// TwinCAT 3 PLC project DPPLC
// Title: YK_DPJ
// Company: YK
// Author: DHW
// ProjectVersion: V1.1
// ProgramVersion: 3.1.4023.0
// CompilerDefines: VISU_USEWSTRING
// libraries:
//   Lib_Basic, * (Beckhoff_GZ)
//   Lib_FileOperation, * (Beckhoff_GZ)
//   Tc2_EtherCAT, * (Beckhoff Automation GmbH)
//   Tc2_Math, * (Beckhoff Automation GmbH)
//   Tc2_MC2, * (Beckhoff Automation GmbH)
//   Tc2_MC2_Camming, * (Beckhoff Automation GmbH)
//   Tc2_MC2_FlyingSaw, * (Beckhoff Automation GmbH)
//   Tc2_Standard, * (Beckhoff Automation GmbH)
//   Tc2_System, * (Beckhoff Automation GmbH)
//   Tc2_TcpIp, * (Beckhoff Automation GmbH)
//   Tc2_Utilities, * (Beckhoff Automation GmbH)
//   Tc2_XmlDataSrv, * (Beckhoff Automation GmbH)
//   Tc3_MC2_AdvancedHoming, * (Beckhoff Automation GmbH)
//   Tc3_Module, * (Beckhoff Automation GmbH)
//   VisuDialogs, * (System)
//   VisuElemEventTable, * (System)
//   VisuSymbols, * (System)
//   VisuSymbols,3.5.10.0,System
// project tree:
//   P2DUTs/01_AxisCO_Ntrol/ MC_AxisParameter.TcDUT, ST_Dust_Motor.TcDUT, ST_ECYCtrl.TcDUT, ST_JXCE.TcDUT, ST_SetpMotor.TcDUT
//   P2DUTs/01_AxisCO_Ntrol_1/ ST_AxisCmd.TcDUT, ST_AxisCtrl.TcDUT, ST_AxisIo.TcDUT, ST_AxisStatus.TcDUT, ST_Axis_Par.TcDUT
//   P2DUTs/02_Cylinder/ ST_CyCmd.TcDUT, ST_CyCtrl.TcDUT, ST_CYIo.TcDUT, ST_CyStatus.TcDUT
//   P2DUTs/06_Interface/FB_Interface/ ST_Cam.TcDUT, ST_Gear.TcDUT, ST_GearInPos.TcDUT, ST_Tension.TcDUT
//   P2DUTs/06_Interface/ IData.TcDUT, IM2Glue.TcDUT
//   P2DUTs/06_Interface/Method/ ST_Method.TcDUT, ST_MethodOut.TcDUT
//   P2DUTs/07_Name/ ST_Dust.TcDUT, ST_AxisName.TcDUT, ST_CylinderName.TcDUT, ST_ElectValveName.TcDUT, ST_P2AxisName.TcDUT, ST_P2CylinderName.TcDUT, ST_P2ElectValveName.TcDUT, ST_P2VirAxisName.TcDUT, ST_RecName.TcDUT, ST_TableName.TcDUT, ST_VirAxisName.TcDUT
//   P2DUTs/08_IO/ ST_Button.TcDUT, ST_P2Button.TcDUT, ST_P2Senser.TcDUT, ST_Senser.TcDUT, ST_SystemButton.TcDUT, System_Senser.TcDUT
//   P2DUTs/30_Parameter/04_Rectify/ ST_PLC_PC_MES.TcDUT, ST_RecCmd.TcDUT, ST_RecCtrl.TcDUT, ST_RecIo.TcDUT, ST_RecStatus.TcDUT
//   P2DUTs/30_Parameter/ ST_DT_To_MQ_MES.TcDUT, ST_MQ_To_DT_MES.TcDUT, ST_ParFilterAD.TcDUT, ST_ParMachine.TcDUT, ST_ParProduct.TcDUT, ST_ParTableNo.TcDUT
//   P2DUTs/31_其他辅助/ DToM_Process.TcDUT, DToM_System.TcDUT, File_com_typ.TcDUT, MToD_Process.TcDUT, MToD_System.TcDUT, ST_DATA_NEED_BE_PERSIS.TcDUT
//   P2DUTs/32_系统/ IModeEN.TcDUT, IRecipe.TcDUT, ST_SysCmd.TcDUT, ST_SystemRUN.TcDUT
//   P2DUTs/33_M2/ ST_BeltData.TcDUT, ST_BeltData1.TcDUT
//   P2DUTs/34_M1/ ST_Rectify.TcDUT
//   P2DUTs/35_CCD/35_CCD/ ICCD_1.TcDUT, STCcdData_1.TcDUT, ST_CCDCom.TcDUT, ST_CCDComOverhang.TcDUT, ST_CCDComRectify.TcDUT, ST_CCDComRectify_I.TcDUT, ST_CCDComRectify_O.TcDUT, ST_CCDOverhang_I.TcDUT, ST_CCDOverhang_O.TcDUT, ST_Ng_classification.TcDUT
//   P2DUTs/35_CCD/ ICCD.TcDUT, STCcdData.TcDUT, STCcdDataSend.TcDUT
//   P2DUTs/36_ShortTest/ CMD.TcDUT, IShortTest.TcDUT, ShortDataShow.TcDUT, ShortPar.TcDUT
//   P2DUTs/37_Code/ ICode.TcDUT, ParCode.TcDUT
//   P2DUTs/38_User1/ ControlSignal.TcDUT, EleControlNo.TcDUT, LocalProduction.TcDUT, P2_AxiseNo.TcDUT, P2_TableNo.TcDUT, Parameters.TcDUT, sMC_CAM_REF.TcDUT, System_Control.TcDUT, User1_Par.TcDUT
//   P2DUTs/39User2/ conAn_date.TcDUT, conCa_date.TcDUT, conDT_Date.TcDUT, conDT_RunStatus.TcDUT, conStickGlue_date.TcDUT, conTailCurl_date.TcDUT, parDT_date.TcDUT, parMechanical.TcDUT, parTailCurl_date.TcDUT, Scan_TJ.TcDUT, ST_Timedata.TcDUT, ST_Torque.TcDUT, ST_UserControl.TcDUT
//   P2DUTs/指纹/ ST_FingerprintKey.TcDUT
//   P2GVLs/ GCylinder.TcGVL, GMotion.TcGVL, GVL_Par.TcGVL, GVL_User2.TcGVL, GVL_User3.TcGVL, IO.TcGVL, N.TcGVL, System.TcGVL, User01.TcGVL
//   P2POUs/BasicFunction/01_IO/ FB_Filter_AD.TcPOU (encrypted, skipped), FB_Filter_ADV2.TcPOU (encrypted, skipped), FB_RotateSwitchCode.TcPOU (encrypted, skipped), ScaleTrans.TcPOU, ScaleTrans_1.TcPOU
//   P2POUs/BasicFunction/02_SystemCheck/ CheckBounds.TcPOU, CheckDivDInt.TcPOU, CheckDivLInt.TcPOU, CheckDivLReal.TcPOU, CheckDivReal.TcPOU, CheckLRangeSigned.TcPOU, CheckLRangeUnsigned.TcPOU, CheckPointer.TcPOU, CheckRangeSigned.TcPOU, CheckRangeUnsigned.TcPOU
//   P2POUs/BasicFunction/03_Motion/ Ax_FindHomeV3.TcPOU (encrypted, skipped), CS_AxisCtrl.TcPOU, CS_DustMoter.TcPOU, CS_SetpMoter.TcPOU, Three_Scale.TcPOU
//   P2POUs/BasicFunction/04_Gear/ FB_GearInDyn.TcPOU (encrypted, skipped), FB_GearInMulti.TcPOU (encrypted, skipped), FB_GearInPos.TcPOU (encrypted, skipped)
//   P2POUs/BasicFunction/05_Actuators/ FB_Cylinder.TcPOU, FB_CylinderV2.TcPOU, FB_Vacuum.TcPOU
//   P2POUs/BasicFunction/06_Public/ FC_AngleToLength.TcPOU (encrypted, skipped), FC_LengthToAngle.TcPOU (encrypted, skipped), f_Length2.TcPOU (encrypted, skipped), f_Length2_1.TcPOU (encrypted, skipped), PulseCtrl.TcPOU (encrypted, skipped), PulseGeneratorCtrl.TcPOU (encrypted, skipped)
//   P2POUs/BasicFunction/07_Ten/ FB_TensionGM.TcPOU (encrypted, skipped), FB_TensionGMV2.TcPOU (encrypted, skipped), FB_TensionGMV2_1.TcPOU (encrypted, skipped), FB_TensionGMV3.TcPOU (encrypted, skipped), FB_TensionP4Buffer.TcPOU (encrypted, skipped), FB_TensionPole.TcPOU (encrypted, skipped), FB_TensionV3.TcPOU (encrypted, skipped)
//   P2POUs/BasicFunction/08_Data/ CS_Data.TcPOU, CS_Data_Test.TcPOU, CS_Recipe.TcPOU, FB_DataXML.TcPOU, FB_DataXML_old.TcPOU, FB_DTData.TcPOU
//   P2POUs/BasicFunction/09_User1/ Dp_Roll_New.TcPOU (encrypted, skipped), Dp_Roll_New_BAK.TcPOU, Dp_Roll_V2.TcPOU, FB_CamIn.TcPOU (encrypted, skipped), FB_CamGMVir.TcPOU (encrypted, skipped), FB_CamPTPTest.TcPOU (encrypted, skipped), FB_CamPTPTestV2.TcPOU (encrypted, skipped), FB_CamTrapezoid.TcPOU (encrypted, skipped), FB_CreatCamEndWind.TcPOU (encrypted, skipped), FB_CreatCamGMBuffer.TcPOU (encrypted, skipped), FB_CreatCamVirGMDriver.TcPOU (encrypted, skipped), FB_CrectCamGMDanserMove.TcPOU (encrypted, skipped), FB_CrectCamMove.TcPOU, FB_CrectCamUpDown.TcPOU, FB_CrectCamUpDown_1.TcPOU, FB_CrectCamUpDown_10.TcPOU, FB_CrectCamUpDown_2.TcPOU, FB_CrectCamUpDown_3.TcPOU, FB_CrectCamUpDown_4.TcPOU, FB_CrectCamYaDaoLine.TcPOU, FB_CrectCamYaDaoLine2_V2.TcPOU, FB_CrectCamYaDaoLine_V2.TcPOU, FB_CrectCamYaDaoUpDown.TcPOU, FB_CrectCamYaDaoUpDown2.TcPOU, FB_GMLengthDown_L.TcPOU (encrypted, skipped), FB_GMLengthDown_R.TcPOU (encrypted, skipped), FB_GMLengthUp.TcPOU (encrypted, skipped), FB_GMLengthUp_L.TcPOU (encrypted, skipped), FB_GMLengthUp_R.TcPOU (encrypted, skipped), FB_RectifyGM.TcPOU (encrypted, skipped)
//   P2POUs/BasicFunction/10_MES/ CS_CcdTcp.TcPOU, CS_CcdTcp_V2.TcPOU, CS_CodeTcp.TcPOU, CS_FsyTcp.TcPOU
//   P2POUs/BasicFunction/11_SystemInfo/ SystemInfoCtrl.TcPOU, TaskInfoCtrl.TcPOU
//   P2POUs/BasicFunction/12_User2/ FB_AxisHandautomatic.TcPOU, FB_BlueFlag.TcPOU, FB_BlueGlue.TcPOU, FB_CamDTDriver.TcPOU, FB_Demarcate.TcPOU, FB_DiameterORLength.TcPOU, FB_RecdevPla.TcPOU, FB_Rectify.TcPOU, FB_RectifyTry.TcPOU, FB_SuckerTest.TcPOU, Program_1.TcPOU, Rectifydev_PID.TcPOU
//   P2POUs/POUS/ FingerprintKey.TcPOU, FunctionTest.TcPOU, IOLink.TcPOU, MAIN.TcPOU, MainState.TcPOU, P2M1_Auto.TcPOU, P2M2_Auto.TcPOU, P2M3_Auto.TcPOU, P2Program_FB.TcPOU
//   P3GVLs/ P3IO.TcGVL, P3Motion.TcGVL, P3Name.TcGVL, P3Par.TcGVL, P3Press.TcGVL, P3Temperature.TcGVL
//   P3POUs/P3FB/ ADSWrite_Limit.TcPOU, CS_AxisCtrlV2.TcPOU (encrypted, skipped), CS_SetpMoterV2.TcPOU, FB_AxisHandautomatic_1.TcPOU, FB_Blink.TcPOU, FB_CSP_Velo_Torque.TcPOU, FB_DataXMLP3.TcPOU, FB_DataXMLP3_Old.TcPOU, FB_HDData.TcPOU, FB_OEE.TcPOU, FB_Press.TcPOU, FB_ProductionDataLocal.TcPOU, FB_PulsPercentage.TcPOU, FB_Temperature.TcPOU, Oven_button.TcPOU, Oven_Time.TcPOU, FB_SetMoter_auto.TcPOU, Sampling.TcPOU, ShortTest.TcPOU, Unwinding_PID.TcPOU, Weight_cese.TcPOU
//   P3POUs/POUs/Auto%28PRG%29/ LateBlanking_Auto1.TcPOU (not stored), LateBlanking_Auto2.TcPOU (not stored), LateBlanking_Auto3.TcPOU (not stored), LateBlanking_Auto4.TcPOU (not stored), LateBlanking_Auto5.TcPOU (not stored), LateBlanking_Auto6.TcPOU (not stored), LateBlanking_Auto7.TcPOU (not stored), LateBlanking_Auto8_01Sticke.TcPOU (not stored), LateBlanking_Auto9_02Sticke.TcPOU (not stored), LateBlanking_Auto1_Stick.TcPOU (not stored)
//   P3POUs/POUs/Auxiliary/ LateBlankingCylinderManual.TcPOU, LateBlankingMotorManual.TcPOU, LateBlanking_Alarm.TcPOU, LateBlanking_Condition.TcPOU, LateBlanking_Scan.TcPOU, LateBlanking_Short_Test.TcPOU, LateBlanking_Temperature.TcPOU, LateBlanking_Thickness_Test.TcPOU, LateBlanking_Tips.TcPOU, LateBlanking_Weight_Test.TcPOU, MES_JT_ZT.TcPOU, MQ_FSY.TcPOU, Output_statistics.TcPOU
//   P3POUs/POUs/Init/ L_Init1.TcPOU, L_Init2.TcPOU, L_Init3.TcPOU, L_Init4.TcPOU, L_Init5.TcPOU, L_Init6.TcPOU, L_Init7.TcPOU, L_Init8.TcPOU
//   P3POUs/POUs/ P3IOLink.TcPOU, P3MAIN.TcPOU, P3MainState.TcPOU
//   P3UDTs/MES/ DTM_Mes1.TcDUT, Mes1.TcDUT, Mes2.TcDUT, MTD_Mes1.TcDUT
//   P3UDTs/Output_statistic/ Statistics.TcDUT, ST_Timedata_1.TcDUT
//   P3UDTs/P3_AxisCO_Ntrol/ ST_AxisCmdV2.TcDUT, ST_AxisCtrlV2.TcDUT, ST_Axis_ParV2.TcDUT
//   P3UDTs/P3_IO/ ST_P3Button.TcDUT, ST_P3Senser.TcDUT
//   P3UDTs/P3_Memory/ ST_CellMemory.TcDUT
//   P3UDTs/P3_Name/ ST_MemoryName.TcDUT, ST_P3AxisName.TcDUT, ST_P3CylinderName.TcDUT, ST_P3ElectValveName.TcDUT, ST_TempName.TcDUT
//   P3UDTs/P3_par/ P3_Par.TcDUT, User2_Par.TcDUT
//   P3UDTs/P3_ShortTest/ CMD_1.TcDUT, ShortCiucitCtrl.TcDUT, ShortDataShow_1.TcDUT, ShortPar_1.TcDUT, ShortTestCtrl.TcDUT, ShortTestReceiveData.TcDUT, ShortTestSendData.TcDUT, ST_ReceiveTestStatus.TcDUT, ST_SendTestStatus.TcDUT
//   P3UDTs/P3_Temperature/ STTempCtrl.TcDUT, ST_ParTemperature.TcDUT, TempIn.TcDUT, TempInShow.TcDUT, TempOut.TcDUT
//   P3UDTs/P3_Thickness/ ST_Thickness.TcDUT
//   P3UDTs/P3_Torque/ ST_TorqueMotion.TcDUT, ST_Torque_P3.TcDUT
//   P3UDTs/P3_Variable/ ST_StickIDGlue_date.TcDUT
//   P3UDTs/P3_Weight/ ST_Gross.TcDUT, ST_ReceiveData.TcDUT, ST_ReceiveStatus.TcDUT, ST_SendData.TcDUT, ST_SendStatus.TcDUT
//   / Task_P2M1.TcTTO, Task_P2M2.TcTTO, Task_P2M3.TcTTO, Task_P2Main.TcTTO, Task_P3.TcTTO
// real-time tasks:
//   TASK Task P1: cycle T#2ms, priority 8, ADS port 350
//   TASK Task P2M1: cycle T#2ms, priority 16, ADS port 351
//   TASK Task P3: cycle T#2ms, priority 18, ADS port 352
//   TASK Task P2M2: cycle T#2ms, priority 14, ADS port 353
//   TASK Task P2M3: cycle T#2ms, priority 12, ADS port 354
//   TASK Task P2Main: cycle T#2ms, priority 10, ADS port 355
// motion (NC):
//   TASK NC-Task 1 SAF: cycle T#2ms, priority 2, ADS port 501
//   TASK NC-Task 1 SVB: cycle T#2ms, priority 4, ADS port 511
//   AXIS Axis001_1 P1An_UnWind_L (id 1) // 正极模切左放卷
//     General: UnitName=°
//     Dynamic: Acceleration=6210, Deceleration=6210, Jerk=225521
//     Velo: SlowManual=20, FastManual=20, Maximum=450
//     OtherSettings: AllowMotionCmdToSlave=true
//     encoder EncType=19
//       EncPara: ScaleFactorNumerator=2.86102e-06, MaxCount=#xffffffff
//     drive DrvType=16
//       DrvPara: MaxCount=#xffffffff, DriveControlDWord=#x00020100
//         Analog: VeloReferenz=450, TorqueSetpointScale=10, ScaleFactorActTorque=0.1
//         TimeComp: TaskDelayCycles=1
//     controller CtrType=1
//       CtrPara: PriorControlFactor=1
//         PosDiffControl: Enable=false
//         Observer: BandWidth=20
//   AXIS Axis002_2 P1An_UnWind_R (id 2) // 正极模切右放卷
//     General: UnitName=°
//     Dynamic: Acceleration=6300, Deceleration=6300, Jerk=220500
//     Velo: SlowManual=20, FastManual=20, Maximum=450
//     OtherSettings: AllowMotionCmdToSlave=true
//     encoder EncType=19
//       EncPara: ScaleFactorNumerator=2.86102e-06, MaxCount=#xffffffff
//     drive DrvType=16
//       DrvPara: MaxCount=#xffffffff, DriveControlDWord=#x00020100
//         Analog: VeloReferenz=450, TorqueSetpointScale=10, ScaleFactorActTorque=0.1
//         TimeComp: TaskDelayCycles=1
//     controller CtrType=1
//       CtrPara: PriorControlFactor=1
//         PosDiffControl: Enable=false
//         Observer: BandWidth=20
//   AXIS Axis003_3 P1An_PoleTension (id 3) // 正极模切前摆杆张力
//     General: UnitName=°
//     Dynamic: Acceleration=120599.992425932, Deceleration=120599.992425932, Jerk=4753059.40298509
//     Velo: FastManual=300, Maximum=9000
//     OtherSettings: AllowMotionCmdToSlave=true
//     encoder EncType=19
//       EncPara: ScaleFactorNumerator=4.29153e-05, Offset=-0.0094842813, MaxCount=#xffffffff, ReferenceSystem=1
//     drive DrvType=16
//       DrvPara: MaxCount=#xffffffff, DriveControlDWord=#x00020000
//         Analog: VeloReferenz=9000, TorqueSetpointScale=10, ScaleFactorActTorque=0.1
//         TimeComp: TaskDelayCycles=1
//     controller CtrType=1
//       CtrPara: PriorControlFactor=1
//         PosDiffControl: Enable=false
//         PID: PosKp=0
//         Observer: BandWidth=20
//   AXIS Axis004_4 P1An_DriverAux (id 4) // 正极模切辅助驱动
//     General: UnitName=°
//     Dynamic: Acceleration=24480, Deceleration=24480, Jerk=924800
//     Velo: SlowManual=20, FastManual=100, Maximum=1800
//     OtherSettings: AllowMotionCmdToSlave=true
//     encoder EncType=19
//       EncPara: ScaleFactorNumerator=8.58307e-06, MaxCount=#xffffffff
//     drive DrvType=16
//       DrvPara: MaxCount=#xffffffff, DriveControlDWord=#x00020100
//         Analog: VeloReferenz=1800, TorqueSetpointScale=10, ScaleFactorActTorque=0.1
//         TimeComp: TaskDelayCycles=1
//     controller CtrType=1
//       CtrPara: PriorControlFactor=1
//         PosDiffControl: Enable=false
//         Observer: BandWidth=20
//   AXIS Axis005_5 P1An_BuffeLine (id 5) // 正极模切极片缓存
//     Dynamic: Acceleration=39520, Deceleration=39520, Jerk=1640580
//     Velo: SlowManual=20, FastManual=20, Maximum=3000
//     OtherSettings: AllowMotionCmdToSlave=true
//     encoder EncType=19
//       EncPara: MaxCount=#xffffffff
//     drive DrvType=16
//       DrvPara: MaxCount=#xffffffff, DriveControlDWord=#x00020100
//         Analog: VeloReferenz=3000, TorqueSetpointScale=10, ScaleFactorActTorque=0.1
//         TimeComp: TaskDelayCycles=1
//     controller CtrType=1
//       CtrPara: PriorControlFactor=1
//         PosDiffControl: Enable=false
//         Observer: BandWidth=20
//   AXIS Axis006_6 P1An_Mould (id 6) // 正极倒角模具
//     General: UnitName=°, UnitFlags=#x00000004
//     Dynamic: Acceleration=50400, Deceleration=50400, Jerk=1764000
//     Velo: SlowManual=10, FastManual=30, Maximum=3600
//     OtherSettings: AllowMotionCmdToSlave=true
//     encoder EncType=19
//       EncPara: ScaleFactorNumerator=8.58307e-06, MaxCount=#xffffffff
//     drive DrvType=16
//       DrvPara: MaxCount=#xffffffff, DriveControlDWord=#x00020100
//         Analog: VeloReferenz=3600, TorqueSetpointScale=10, ScaleFactorActTorque=0.1
//         TimeComp: TaskDelayCycles=1
//     controller CtrType=1
//       CtrPara: PriorControlFactor=1
//         PosDiffControl: Enable=false
//         Observer: BandWidth=20
//   AXIS Axis007_7 P1An_MouldRectify_X (id 7) // 正极模具纠偏X轴(肩宽)
//     Dynamic: Acceleration=3875, Deceleration=3875, Jerk=109205
//     Velo: SlowManual=20, FastManual=20, Maximum=250
//     OtherSettings: AllowMotionCmdToSlave=true
//     encoder EncType=19
//       EncPara: ScaleFactorNumerator=5.96046e-07, MaxCount=#xffffffff
//     drive DrvType=16
//       DrvPara: MaxCount=#xffffffff, DriveControlDWord=#x00020100
//         Analog: VeloReferenz=250, TorqueSetpointScale=10, ScaleFactorActTorque=0.1
//         TimeComp: TaskDelayCycles=1
//     controller CtrType=1
//       CtrPara: PriorControlFactor=1
//         Observer: BandWidth=20
//   AXIS Axis008_8 P1An_MouldRectify_Y (id 8) // 正极模具纠偏Y轴(切刀深度)
//     Dynamic: Acceleration=450, Deceleration=450, Jerk=1620
//     Velo: SlowManual=20, FastManual=20, Maximum=250
//     OtherSettings: AllowMotionCmdToSlave=true
//     encoder EncType=19
//       EncPara: ScaleFactorNumerator=5.96046e-07, MaxCount=#xffffffff
//     drive DrvType=16
//       DrvPara: MaxCount=#xffffffff, DriveControlDWord=#x00020100
//         Analog: VeloReferenz=250, TorqueSetpointScale=10, ScaleFactorActTorque=0.1
//         TimeComp: TaskDelayCycles=1
//     controller CtrType=1
//       CtrPara: PriorControlFactor=1
//         PosDiffControl: Enable=false
//         Observer: BandWidth=20
//   AXIS Axis009_9 P1An_DriverDDR (id 9) // 正极模切主驱动
//     General: UnitName=°
//     Dynamic: Acceleration=42582, Deceleration=42582, Jerk=1260760
//     Velo: SlowManual=20, FastManual=20, Maximum=2820
//     OtherSettings: AllowMotionCmdToSlave=true
//     encoder EncType=19
//       EncPara: ScaleFactorNumerator=0.001, MaxCount=#xffffffff
//     drive DrvType=16
//       DrvPara: MaxCount=#xffffffff, DriveControlDWord=#x00020100
//         Analog: VeloReferenz=2820, TorqueSetpointScale=10, ScaleFactorActTorque=0.1
//         TimeComp: TaskDelayCycles=1
//     controller CtrType=1
//       CtrPara: PriorControlFactor=1
//         Observer: BandWidth=20
//   AXIS Axis010_10 P1An_Cuter (id 10) // 正极裁切切刀
//     General: UnitName=°, UnitFlags=#x00000004
//     Dynamic: Acceleration=48960, Deceleration=48960, Jerk=1849600
//     Velo: SlowManual=20, FastManual=20, Maximum=3600
//     OtherSettings: ErrorReactionMode=1, ErrorReactionDelay=1000, AllowMotionCmdToSlave=true
//     encoder EncType=19
//       EncPara: ScaleFactorNumerator=8.58307e-06, MaxCount=#xffffffff
//     drive DrvType=16
//       DrvPara: MaxCount=#xffffffff, DriveControlDWord=#x00020100
//         Analog: VeloReferenz=3600, TorqueSetpointScale=10, ScaleFactorActTorque=0.1
//         TimeComp: TaskDelayCycles=1
//     controller CtrType=1
//       CtrPara: PriorControlFactor=1
//         PosDiffControl: Enable=false
//         Observer: BandWidth=20
//   AXIS Axis011_11 P1An_CuterDegRectify (id 11) // 正极裁切角度纠偏
//     General: UnitName=°
//     Dynamic: Acceleration=271.999960582622, Deceleration=271.999960582622, Jerk=10275.5970217855
//     Velo: SlowManual=20, FastManual=20, Maximum=20
//     OtherSettings: ErrorReactionMode=1, ErrorReactionDelay=1000, AllowMotionCmdToSlave=true
//     encoder EncType=19
//       EncPara: ScaleFactorNumerator=4.85275e-08, Inverse=true, MaxCount=#xffffffff
//     drive DrvType=16
//       DrvPara: Inverse=true, MaxCount=#xffffffff, DriveControlDWord=#x00020100
//         Analog: VeloReferenz=20, TorqueSetpointScale=10, ScaleFactorActTorque=0.1
//         TimeComp: TaskDelayCycles=1
//     controller CtrType=1
//       CtrPara: PriorControlFactor=1
//         Observer: BandWidth=20
//   AXIS Axis012_12 P1An_CuterBelt (id 12) // 正极裁切输送皮带
//     Dynamic: Acceleration=30140.0335128451, Deceleration=30140.0335128451, Jerk=1115992.4817532
//     Velo: SlowManual=20, FastManual=20, Maximum=2200
//     OtherSettings: AllowMotionCmdToSlave=true
//     encoder EncType=19
//       EncPara: ScaleFactorNumerator=5.3929e-06, MaxCount=#xffffffff
//     drive DrvType=16
//       DrvPara: MaxCount=#xffffffff, DriveControlDWord=#x00020100
//         Analog: TorqueSetpointScale=10, ScaleFactorActTorque=0.1
//         TimeComp: TaskDelayCycles=1
//     controller CtrType=1
//       CtrPara: PriorControlFactor=1
//         PosDiffControl: Enable=false
//         Observer: BandWidth=20
//   AXIS Axis013_13 P1An_CuterBeltChange (id 13) // 正极裁切输送带换型
//     Dynamic: Acceleration=3400, Deceleration=3400, Jerk=128444
//     Velo: SlowManual=3, FastManual=3, Maximum=250
//     OtherSettings: AllowMotionCmdToSlave=true
//     encoder EncType=19
//       EncPara: ScaleFactorNumerator=5.96046e-07, Offset=-2.8610208e-05, MaxCount=#xffffffff, ReferenceSystem=1
//     drive DrvType=16
//       DrvPara: MaxCount=#xffffffff, DriveControlDWord=#x00020100
//         Analog: VeloReferenz=250, TorqueSetpointScale=10, ScaleFactorActTorque=0.1
//         TimeComp: TaskDelayCycles=1
//     controller CtrType=1
//       CtrPara: PriorControlFactor=1
//         Observer: BandWidth=20
//   AXIS Axis014_14 P1An_CCDPressPush (id 14) // 正极尺寸CCD压片升降
//     General: UnitName=°, UnitFlags=#x00000004
//     Dynamic: Acceleration=48600.0096022021, Deceleration=48600.0096022021, Jerk=1874570.74074081
//     Velo: SlowManual=20, FastManual=20, Maximum=3600
//     OtherSettings: AllowMotionCmdToSlave=true
//     encoder EncType=19
//       EncPara: ScaleFactorNumerator=8.58307e-06, MaxCount=#xffffffff
//     drive DrvType=16
//       DrvPara: MaxCount=#xffffffff, DriveControlDWord=#x00020100
//         Analog: VeloReferenz=3600, TorqueSetpointScale=10, ScaleFactorActTorque=0.1
//         TimeComp: TaskDelayCycles=1
//     controller CtrType=1
//       CtrPara: PriorControlFactor=1
//         PosDiffControl: Enable=false
//         Observer: BandWidth=20
//   AXIS Axis015_15 P1An_NGPushReverseBelt (id 15) // 正极踢废倒装皮带
//     Dynamic: Acceleration=38181.0021027927, Deceleration=38181.0021027927, Jerk=1269740.13986014
//     Velo: SlowManual=5, FastManual=10, Maximum=2670
//     OtherSettings: AllowMotionCmdToSlave=true
//     encoder EncType=19
//       EncPara: ScaleFactorNumerator=6.51642e-06, MaxCount=#xffffffff
//     drive DrvType=16
//       DrvPara: MaxCount=#xffffffff, DriveControlDWord=#x00020100
//         Analog: VeloReferenz=2670, TorqueSetpointScale=10, ScaleFactorActTorque=0.1
//         TimeComp: TaskDelayCycles=1
//     controller CtrType=1
//       CtrPara: PriorControlFactor=1
//         PosDiffControl: Enable=false
//         Observer: BandWidth=20
//   AXIS Axis016_16 P1An_NGPush1 (id 16) // 正极踢连续废料
//     General: UnitName=°, UnitFlags=#x00000004
//     Dynamic: Acceleration=248400.015963037, Deceleration=248400.015963037, Jerk=9020841.15942032
//     Velo: SlowManual=5, FastManual=10, Maximum=18000
//     OtherSettings: AllowMotionCmdToSlave=true
//     encoder EncType=19
//       EncPara: ScaleFactorNumerator=4.29153e-05, MaxCount=#xffffffff
//     drive DrvType=16
//       DrvPara: MaxCount=#xffffffff, DriveControlDWord=#x00020100
//         Analog: VeloReferenz=18000, TorqueSetpointScale=10, ScaleFactorActTorque=0.1
//         TimeComp: TaskDelayCycles=1
//     controller CtrType=1
//       CtrPara: PriorControlFactor=1
//         PosDiffControl: Enable=false
//         Observer: BandWidth=20
//   AXIS Axis017_17 P1An_NGPush2 (id 17) // 正极踢单张废料
//     General: UnitName=°, UnitFlags=#x00000004
//     Dynamic: Acceleration=21120, Deceleration=21120, Jerk=871200
//     Velo: SlowManual=5, FastManual=10, Maximum=1600
//     OtherSettings: AllowMotionCmdToSlave=true
//     encoder EncType=19
//       EncPara: ScaleFactorNumerator=4.29153e-05, MaxCount=#xffffffff
//     drive DrvType=16
//       DrvPara: MaxCount=#xffffffff, DriveControlDWord=#x00020100
//         Analog: VeloReferenz=1800, TorqueSetpointScale=10, ScaleFactorActTorque=0.1
//         TimeComp: TaskDelayCycles=1
//     controller CtrType=1
//       CtrPara: PriorControlFactor=1
//         PosDiffControl: Enable=false
//         Observer: BandWidth=20
//   AXIS Axis018_18 P1An_DedustBelt (id 18) // 正极上表面除尘皮带
//     Dynamic: Acceleration=37914.0374926863, Deceleration=37914.0374926863, Jerk=1281852.53521252
//     Velo: SlowManual=20, FastManual=20, Maximum=2670
//     OtherSettings: AllowMotionCmdToSlave=true
//     encoder EncType=19
//       EncPara: ScaleFactorNumerator=6.51642e-06, MaxCount=#xffffffff
//     drive DrvType=16
//       DrvPara: MaxCount=#xffffffff, DriveControlDWord=#x00020100
//         Analog: VeloReferenz=2670, TorqueSetpointScale=10, ScaleFactorActTorque=0.1
//         TimeComp: TaskDelayCycles=1
//     controller CtrType=1
//       CtrPara: PriorControlFactor=1
//         PosDiffControl: Enable=false
//         Observer: BandWidth=20
//   AXIS Axis019_19 P1An_DedustReverseBelt (id 19) // 正极下表面除尘倒装皮带
//     Dynamic: Acceleration=36045.0168406667, Deceleration=36045.0168406667, Jerk=1390311.29914012
//     Velo: SlowManual=20, FastManual=20, Maximum=2670
//     OtherSettings: AllowMotionCmdToSlave=true
//     encoder EncType=19
//       EncPara: ScaleFactorNumerator=6.51642e-06, MaxCount=#xffffffff
//     drive DrvType=16
//       DrvPara: MaxCount=#xffffffff, DriveControlDWord=#x00020100
//         Analog: VeloReferenz=2670, TorqueSetpointScale=10, ScaleFactorActTorque=0.1
//         TimeComp: TaskDelayCycles=1
//     controller CtrType=1
//       CtrPara: PriorControlFactor=1
//         PosDiffControl: Enable=false
//         Observer: BandWidth=20
//   AXIS Axis020_20 P1An_SubBelt1 (id 20) // 正极送料分段皮带1
//     Dynamic: Acceleration=34100, Deceleration=34100, Jerk=1571360
//     Velo: SlowManual=20, FastManual=100, Maximum=2670
//     OtherSettings: AllowMotionCmdToSlave=true
//     encoder EncType=19
//       EncPara: ScaleFactorNumerator=6.51642e-06, MaxCount=#xffffffff
//     drive DrvType=16
//       DrvPara: MaxCount=#xffffffff, DriveControlDWord=#x00020100
//         Analog: VeloReferenz=2670, TorqueSetpointScale=10, ScaleFactorActTorque=0.1
//         TimeComp: TaskDelayCycles=1
//     controller CtrType=1
//       CtrPara: PriorControlFactor=1
//         PosDiffControl: Enable=false
//         Observer: BandWidth=20
//   AXIS Axis021_21 P1An_SubBelt2 (id 21) // 正极送料分段皮带2
//     Dynamic: Acceleration=37113, Deceleration=37113, Jerk=1322750
//     Velo: FastManual=200, Maximum=2670
//     OtherSettings: AllowMotionCmdToSlave=true
//     encoder EncType=19
//       EncPara: ScaleFactorNumerator=6.51642e-06, MaxCount=#xffffffff
//     drive DrvType=16
//       DrvPara: MaxCount=#xffffffff, DriveControlDWord=#x00020100
//         Analog: VeloReferenz=2670, TorqueSetpointScale=10, ScaleFactorActTorque=0.1
//         TimeComp: TaskDelayCycles=1
//     controller CtrType=1
//       CtrPara: PriorControlFactor=1
//         PosDiffControl: Enable=false
//         Observer: BandWidth=20
//   AXIS Axis022_22 P1An_SubBelt3 (id 22) // 正极送料分段皮带3
//     Dynamic: Acceleration=34100, Deceleration=34100, Jerk=1571360
//     Velo: SlowManual=20, FastManual=100, Maximum=2670
//     OtherSettings: AllowMotionCmdToSlave=true
//     encoder EncType=19
//       EncPara: ScaleFactorNumerator=6.51642e-06, MaxCount=#xffffffff
//     drive DrvType=16
//       DrvPara: MaxCount=#xffffffff, DriveControlDWord=#x00020100
//         Analog: VeloReferenz=2670, TorqueSetpointScale=10, ScaleFactorActTorque=0.1
//         TimeComp: TaskDelayCycles=1
//     controller CtrType=1
//       CtrPara: PriorControlFactor=1
//         PosDiffControl: Enable=false
//         Observer: BandWidth=20
//   AXIS Axis023_23 P1An_Ready1 (id 23) // P1备用1
//     Dynamic: Acceleration=25013.3, Deceleration=25013.3, Jerk=657214
//     Velo: FastManual=300, Maximum=4100
//     OtherSettings: AllowMotionCmdToSlave=true
//     encoder EncType=1
//       EncPara: ScaleFactorNumerator=9.93411e-06, ModuloFactor=114.59156
//     drive DrvType=5
//       Analog: VeloReferenz=4300, TorqueSetpointScale=10, ScaleFactorActTorque=0.1
//       TimeComp: TaskDelayCycles=1
//     controller CtrType=1
//       CtrPara: PriorControlFactor=1
//         PosDiffControl: Enable=false
//         PID: PosKp=0
//         Observer: BandWidth=20
//   AXIS Axis024_24 P1An_Ready2 (id 24) // P1备用2
//     General: UnitName=°, UnitFlags=#x00000004
//     Dynamic: Acceleration=34109.1, Deceleration=34109.1, Jerk=1222090
//     Velo: SlowManual=20, FastManual=100, Maximum=18000
//     OtherSettings: AllowMotionCmdToSlave=true
//     encoder EncType=1
//       EncPara: ScaleFactorNumerator=4.29153e-05
//     drive DrvType=5
//       Analog: VeloReferenz=20000, TorqueSetpointScale=10, ScaleFactorActTorque=0.1
//       TimeComp: TaskDelayCycles=1
//     controller CtrType=1
//       CtrPara: PriorControlFactor=1
//         PosDiffControl: Enable=false
//         Observer: BandWidth=20
//   AXIS Axis025_25 P1Ca_UnWind_L (id 25) // 负极模切左放卷
//     General: UnitName=°
//     Dynamic: Acceleration=6029.9996212966, Deceleration=6029.9996212966, Jerk=237652.970149255
//     Velo: SlowManual=20, FastManual=100, Maximum=450
//     OtherSettings: AllowMotionCmdToSlave=true
//     encoder EncType=19
//       EncPara: ScaleFactorNumerator=2.86102e-06, MaxCount=#xffffffff
//     drive DrvType=16
//       DrvPara: MaxCount=#xffffffff, DriveControlDWord=#x00020100
//         Analog: VeloReferenz=450, TorqueSetpointScale=10, ScaleFactorActTorque=0.1
//         TimeComp: TaskDelayCycles=1
//     controller CtrType=1
//       CtrPara: PriorControlFactor=1
//         PosDiffControl: Enable=false
//         Observer: BandWidth=20
//   AXIS Axis026_26 P1Ca_UnWind_R (id 26) // 负极模切右放卷
//     General: UnitName=°
//     Dynamic: Acceleration=6254.99697221163, Deceleration=6254.99697221163, Jerk=222934.784172714
//     Velo: SlowManual=20, FastManual=100, Maximum=450
//     OtherSettings: AllowMotionCmdToSlave=true
//     encoder EncType=19
//       EncPara: ScaleFactorNumerator=2.86102e-06, MaxCount=#xffffffff
//     drive DrvType=16
//       DrvPara: MaxCount=#xffffffff, DriveControlDWord=#x00020100
//         Analog: VeloReferenz=450, TorqueSetpointScale=10, ScaleFactorActTorque=0.1
//         TimeComp: TaskDelayCycles=1
//     controller CtrType=1
//       CtrPara: PriorControlFactor=1
//         PosDiffControl: Enable=false
//         Observer: BandWidth=20
//   AXIS Axis027_27 P1Ca_PoleTension (id 27) // 负极模切前摆杆张力
//     General: UnitName=°
//     Dynamic: Acceleration=120599.992425932, Deceleration=120599.992425932, Jerk=4753059.40298509
//     Velo: FastManual=300, Maximum=9000
//     OtherSettings: AllowMotionCmdToSlave=true
//     encoder EncType=19
//       EncPara: ScaleFactorNumerator=4.29153e-05, Offset=-0.0503396469, ModuloFactor=114.59156, MaxCount=#xffffffff, ReferenceSystem=1
//     drive DrvType=16
//       DrvPara: MaxCount=#xffffffff, DriveControlDWord=#x00020000
//         Analog: VeloReferenz=9000, TorqueSetpointScale=10, ScaleFactorActTorque=0.1
//         TimeComp: TaskDelayCycles=1
//     controller CtrType=1
//       CtrPara: PriorControlFactor=1
//         PosDiffControl: Enable=false
//         PID: PosKp=0
//         Observer: BandWidth=20
//   AXIS Axis028_28 P1Ca_DriverAux (id 28) // 负极模切辅助驱动
//     General: UnitName=°
//     Dynamic: Acceleration=24840.0015963037, Deceleration=24840.0015963037, Jerk=902084.115942032
//     Velo: SlowManual=20, FastManual=100, Maximum=1800
//     OtherSettings: AllowMotionCmdToSlave=true
//     encoder EncType=19
//       EncPara: ScaleFactorNumerator=8.58307e-06, MaxCount=#xffffffff
//     drive DrvType=16
//       DrvPara: MaxCount=#xffffffff, DriveControlDWord=#x00020100
//         Analog: VeloReferenz=1800, TorqueSetpointScale=10, ScaleFactorActTorque=0.1
//         TimeComp: TaskDelayCycles=1
//     controller CtrType=1
//       CtrPara: PriorControlFactor=1
//         PosDiffControl: Enable=false
//         Observer: BandWidth=20
//   AXIS Axis029_29 P1Ca_BuffeLine (id 29) // 负极模切极片缓存
//     Dynamic: Acceleration=41400.0279353762, Deceleration=41400.0279353762, Jerk=1503472.02898619
//     Velo: SlowManual=20, FastManual=100, Maximum=3000
//     OtherSettings: AllowMotionCmdToSlave=true
//     encoder EncType=19
//       EncPara: MaxCount=#xffffffff
//     drive DrvType=16
//       DrvPara: MaxCount=#xffffffff, DriveControlDWord=#x00020100
//         Analog: VeloReferenz=3000, TorqueSetpointScale=10, ScaleFactorActTorque=0.1
//         TimeComp: TaskDelayCycles=1
//     controller CtrType=1
//       CtrPara: PriorControlFactor=1
//         PosDiffControl: Enable=false
//         Observer: BandWidth=20
//   AXIS Axis030_30 P1Ca_Mould (id 30) // 负极倒角模具
//     General: UnitName=°, UnitFlags=#x00000004
//     Dynamic: Acceleration=49320.0216847281, Deceleration=49320.0216847281, Jerk=1826171.60583977
//     Velo: Maximum=3600
//     OtherSettings: AllowMotionCmdToSlave=true
//     encoder EncType=19
//       EncPara: ScaleFactorNumerator=8.58307e-06, MaxCount=#xffffffff
//     drive DrvType=16
//       DrvPara: MaxCount=#xffffffff, DriveControlDWord=#x00020100
//         Analog: VeloReferenz=3600, TorqueSetpointScale=10, ScaleFactorActTorque=0.1
//         TimeComp: TaskDelayCycles=1
//     controller CtrType=1
//       CtrPara: PriorControlFactor=1
//         PosDiffControl: Enable=false
//         Observer: BandWidth=20
//   AXIS Axis031_31 P1Ca_MouldRectify_X (id 31) // 负极模具纠偏X轴(肩宽)
//     Dynamic: Acceleration=3400.00311419763, Deceleration=3400.00311419763, Jerk=128444.235294225
//     Velo: Maximum=250
//     OtherSettings: AllowMotionCmdToSlave=true
//     encoder EncType=19
//       EncPara: ScaleFactorNumerator=5.96046e-07, MaxCount=#xffffffff
//     drive DrvType=16
//       DrvPara: MaxCount=#xffffffff, DriveControlDWord=#x00020100
//         Analog: VeloReferenz=250, TorqueSetpointScale=10, ScaleFactorActTorque=0.1
//         TimeComp: TaskDelayCycles=1
//     controller CtrType=1
//       CtrPara: PriorControlFactor=1
//         Observer: BandWidth=20
//   AXIS Axis032_32 P1Ca_MouldRectify_Y (id 32) // 负极模具纠偏Y轴(切刀深度)
//     Dynamic: Acceleration=3500, Deceleration=3500, Jerk=122500
//     Velo: Maximum=250
//     OtherSettings: AllowMotionCmdToSlave=true
//     encoder EncType=19
//       EncPara: ScaleFactorNumerator=5.96046e-07, MaxCount=#xffffffff
//     drive DrvType=16
//       DrvPara: MaxCount=#xffffffff, DriveControlDWord=#x00020100
//         Analog: VeloReferenz=250, TorqueSetpointScale=10, ScaleFactorActTorque=0.1
//         TimeComp: TaskDelayCycles=1
//     controller CtrType=1
//       CtrPara: PriorControlFactor=1
//         PosDiffControl: Enable=false
//         Observer: BandWidth=20
//   AXIS Axis033_33 P1Ca_DriverDDR (id 33) // 负极模切主驱动
//     General: UnitName=°
//     Dynamic: Acceleration=39198.0149757196, Deceleration=39198.0149757196, Jerk=1397061.06750257
//     Velo: Maximum=2820
//     OtherSettings: AllowMotionCmdToSlave=true
//     encoder EncType=19
//       EncPara: ScaleFactorNumerator=0.001, MaxCount=#xffffffff
//     drive DrvType=16
//       DrvPara: MaxCount=#xffffffff, DriveControlDWord=#x00020100
//         Analog: VeloReferenz=2820, TorqueSetpointScale=10, ScaleFactorActTorque=0.1
//         TimeComp: TaskDelayCycles=1
//     controller CtrType=1
//       CtrPara: PriorControlFactor=1
//         Observer: BandWidth=20
//   AXIS Axis034_34 P1Ca_Cuter (id 34) // 负极裁切切刀
//     General: UnitName=°, UnitFlags=#x00000004
//     Dynamic: Acceleration=49679.9880277357, Deceleration=49679.9880277357, Jerk=1804169.13043489
//     Velo: Maximum=3600
//     OtherSettings: AllowMotionCmdToSlave=true
//     encoder EncType=19
//       EncPara: ScaleFactorNumerator=8.58307e-06, MaxCount=#xffffffff
//     drive DrvType=16
//       DrvPara: MaxCount=#xffffffff, DriveControlDWord=#x00020100
//         Analog: VeloReferenz=3600, TorqueSetpointScale=10, ScaleFactorActTorque=0.1
//         TimeComp: TaskDelayCycles=1
//     controller CtrType=1
//       CtrPara: PriorControlFactor=1
//         PosDiffControl: Enable=false
//         Observer: BandWidth=20
//   AXIS Axis035_35 P1Ca_CuterDegRectify (id 35) // 负极裁切角度纠偏
//     General: UnitName=°
//     Dynamic: Acceleration=281.999989688649, Deceleration=281.999989688649, Jerk=9698.04929078015
//     Velo: Maximum=20
//     OtherSettings: AllowMotionCmdToSlave=true
//     encoder EncType=19
//       EncPara: ScaleFactorNumerator=4.85275e-08, MaxCount=#xffffffff
//     drive DrvType=16
//       DrvPara: MaxCount=#xffffffff, DriveControlDWord=#x00020100
//         Analog: VeloReferenz=20, TorqueSetpointScale=10, ScaleFactorActTorque=0.1
//         TimeComp: TaskDelayCycles=1
//     controller CtrType=1
//       CtrPara: PriorControlFactor=1
//         Observer: BandWidth=20
//   AXIS Axis036_36 P1Ca_CuterBelt (id 36) // 负极裁切输送皮带
//     Dynamic: Acceleration=30360.0104062668, Deceleration=30360.0104062668, Jerk=1102550.75582552
//     Velo: Maximum=2200
//     OtherSettings: AllowMotionCmdToSlave=true
//     encoder EncType=19
//       EncPara: ScaleFactorNumerator=5.3929e-06, MaxCount=#xffffffff
//     drive DrvType=16
//       DrvPara: MaxCount=#xffffffff, DriveControlDWord=#x00020100
//         Analog: TorqueSetpointScale=10, ScaleFactorActTorque=0.1
//         TimeComp: TaskDelayCycles=1
//     controller CtrType=1
//       CtrPara: PriorControlFactor=1
//         PosDiffControl: Enable=false
//         Observer: BandWidth=20
//   AXIS Axis037_37 P1Ca_CuterBeltChange (id 37) // 负极裁切输送带换型
//     Dynamic: Acceleration=3574.9993694312, Deceleration=3574.9993694312, Jerk=118889.958059682
//     Velo: FastManual=200, Maximum=250
//     OtherSettings: ErrorReactionMode=1, ErrorReactionDelay=1000, AllowMotionCmdToSlave=true
//     encoder EncType=19
//       EncPara: ScaleFactorNumerator=5.96046e-07, Offset=2.384184e-06, MaxCount=#xffffffff, ReferenceSystem=1
//     drive DrvType=16
//       DrvPara: MaxCount=#xffffffff, DriveControlDWord=#x00020100
//         Analog: VeloReferenz=250, TorqueSetpointScale=10, ScaleFactorActTorque=0.1
//         TimeComp: TaskDelayCycles=1
//     controller CtrType=1
//       CtrPara: PriorControlFactor=1
//         Observer: BandWidth=20
//   AXIS Axis038_38 P1Ca_CCDPressPush (id 38) // 负极尺寸CCD压片升降
//     General: UnitName=°, UnitFlags=#x00000004
//     Dynamic: Acceleration=47879.9944033041, Deceleration=47879.9944033041, Jerk=1929709.54887221
//     Velo: FastManual=200, Maximum=3600
//     OtherSettings: ErrorReactionMode=1, ErrorReactionDelay=1000, AllowMotionCmdToSlave=true
//     encoder EncType=19
//       EncPara: ScaleFactorNumerator=8.58307e-06, MaxCount=#xffffffff
//     drive DrvType=16
//       DrvPara: MaxCount=#xffffffff, DriveControlDWord=#x00020100
//         Analog: VeloReferenz=3600, TorqueSetpointScale=10, ScaleFactorActTorque=0.1
//         TimeComp: TaskDelayCycles=1
//     controller CtrType=1
//       CtrPara: PriorControlFactor=1
//         PosDiffControl: Enable=false
//         Observer: BandWidth=20
//   AXIS Axis039_39 P1Ca_NGPushReverseBelt (id 39) // 负极踢废倒装皮带
//     Dynamic: Acceleration=36312.0129556683, Deceleration=36312.0129556683, Jerk=1371790.97887527
//     Velo: FastManual=200, Maximum=2670
//     OtherSettings: AllowMotionCmdToSlave=true
//     encoder EncType=19
//       EncPara: ScaleFactorNumerator=6.51642e-06, MaxCount=#xffffffff
//     drive DrvType=16
//       DrvPara: MaxCount=#xffffffff, DriveControlDWord=#x00020100
//         Analog: VeloReferenz=2670, TorqueSetpointScale=10, ScaleFactorActTorque=0.1
//         TimeComp: TaskDelayCycles=1
//     controller CtrType=1
//       CtrPara: PriorControlFactor=1
//         PosDiffControl: Enable=false
//         Observer: BandWidth=20
//   AXIS Axis040_40 P1Ca_NGPush1 (id 40) // 负极踢连续废料
//     General: UnitName=°, UnitFlags=#x00000004
//     Dynamic: Acceleration=242999.980795616, Deceleration=242999.980795616, Jerk=9372858.51851857
//     Velo: FastManual=200, Maximum=18000
//     OtherSettings: AllowMotionCmdToSlave=true
//     encoder EncType=19
//       EncPara: ScaleFactorNumerator=4.29153e-05, MaxCount=#xffffffff
//     drive DrvType=16
//       DrvPara: MaxCount=#xffffffff, DriveControlDWord=#x00020100
//         Analog: VeloReferenz=18000, TorqueSetpointScale=10, ScaleFactorActTorque=0.1
//         TimeComp: TaskDelayCycles=1
//     controller CtrType=1
//       CtrPara: PriorControlFactor=1
//         PosDiffControl: Enable=false
//         Observer: BandWidth=20
//   AXIS Axis041_41 P1Ca_NGPush2 (id 41) // 负极踢单张废料
//     General: UnitName=°, UnitFlags=#x00000004
//     Dynamic: Acceleration=246600.035484062, Deceleration=246600.035484062, Jerk=9130862.62773741
//     Velo: FastManual=200, Maximum=18000
//     OtherSettings: AllowMotionCmdToSlave=true
//     encoder EncType=19
//       EncPara: ScaleFactorNumerator=4.29153e-05, MaxCount=#xffffffff
//     drive DrvType=16
//       DrvPara: MaxCount=#xffffffff, DriveControlDWord=#x00020100
//         Analog: VeloReferenz=18000, TorqueSetpointScale=10, ScaleFactorActTorque=0.1
//         TimeComp: TaskDelayCycles=1
//     controller CtrType=1
//       CtrPara: PriorControlFactor=1
//         PosDiffControl: Enable=false
//         Observer: BandWidth=20
//   AXIS Axis042_42 P1Ca_DedustBelt (id 42) // 负极上表面除尘皮带
//     Dynamic: Acceleration=36045.0168406667, Deceleration=36045.0168406667, Jerk=1390311.29914012
//     Velo: FastManual=200, Maximum=2670
//     OtherSettings: AllowMotionCmdToSlave=true
//     encoder EncType=19
//       EncPara: ScaleFactorNumerator=6.51642e-06, MaxCount=#xffffffff
//     drive DrvType=16
//       DrvPara: MaxCount=#xffffffff, DriveControlDWord=#x00020100
//         Analog: VeloReferenz=2670, TorqueSetpointScale=10, ScaleFactorActTorque=0.1
//         TimeComp: TaskDelayCycles=1
//     controller CtrType=1
//       CtrPara: PriorControlFactor=1
//         PosDiffControl: Enable=false
//         Observer: BandWidth=20
//   AXIS Axis043_43 P1Ca_DedustReverseBelt (id 43) // 负极下表面除尘倒装皮带
//     Dynamic: Acceleration=35778.0265093222, Deceleration=35778.0265093222, Jerk=1410072.08955301
//     Velo: FastManual=200, Maximum=2670
//     OtherSettings: AllowMotionCmdToSlave=true
//     encoder EncType=19
//       EncPara: ScaleFactorNumerator=6.51642e-06, MaxCount=#xffffffff
//     drive DrvType=16
//       DrvPara: MaxCount=#xffffffff, DriveControlDWord=#x00020100
//         Analog: VeloReferenz=2670, TorqueSetpointScale=10, ScaleFactorActTorque=0.1
//         TimeComp: TaskDelayCycles=1
//     controller CtrType=1
//       CtrPara: PriorControlFactor=1
//         PosDiffControl: Enable=false
//         Observer: BandWidth=20
//   AXIS Axis044_44 P1Ca_SubBelt1 (id 44) // 负极送料分段皮带1
//     Dynamic: Acceleration=36579.0118280284, Deceleration=36579.0118280284, Jerk=1354410.87591255
//     Velo: SlowManual=5, FastManual=10, Maximum=2670
//     OtherSettings: AllowMotionCmdToSlave=true
//     encoder EncType=19
//       EncPara: ScaleFactorNumerator=6.51642e-06, MaxCount=#xffffffff
//     drive DrvType=16
//       DrvPara: MaxCount=#xffffffff, DriveControlDWord=#x00020100
//         Analog: VeloReferenz=2670, TorqueSetpointScale=10, ScaleFactorActTorque=0.1
//         TimeComp: TaskDelayCycles=1
//     controller CtrType=1
//       CtrPara: PriorControlFactor=1
//         PosDiffControl: Enable=false
//         Observer: BandWidth=20
//   AXIS Axis045_45 P1Ca_SubBelt2 (id 45) // 负极送料分段皮带2
//     Dynamic: Acceleration=37646.9958754605, Deceleration=37646.9958754605, Jerk=1294689.71631207
//     Velo: SlowManual=5, FastManual=10, Maximum=2670
//     OtherSettings: AllowMotionCmdToSlave=true
//     encoder EncType=19
//       EncPara: ScaleFactorNumerator=6.51642e-06, MaxCount=#xffffffff
//     drive DrvType=16
//       DrvPara: MaxCount=#xffffffff, DriveControlDWord=#x00020100
//         Analog: VeloReferenz=2670, TorqueSetpointScale=10, ScaleFactorActTorque=0.1
//         TimeComp: TaskDelayCycles=1
//     controller CtrType=1
//       CtrPara: PriorControlFactor=1
//         PosDiffControl: Enable=false
//         Observer: BandWidth=20
//   AXIS Axis046_46 P1Ca_SubBelt3 (id 46) // 负极送料分段皮带3
//     Dynamic: Acceleration=37913.9879241294, Deceleration=37913.9879241294, Jerk=1281859.18343762
//     Velo: Maximum=2670
//     OtherSettings: AllowMotionCmdToSlave=true
//     encoder EncType=19
//       EncPara: ScaleFactorNumerator=6.51642e-06, MaxCount=#xffffffff
//     drive DrvType=16
//       DrvPara: MaxCount=#xffffffff, DriveControlDWord=#x00020100
//         Analog: VeloReferenz=2670, TorqueSetpointScale=10, ScaleFactorActTorque=0.1
//         TimeComp: TaskDelayCycles=1
//     controller CtrType=1
//       CtrPara: PriorControlFactor=1
//         PosDiffControl: Enable=false
//         Observer: BandWidth=20
//   AXIS Axis047_47 P1Ca_Ready1 (id 47) // P2备用1
//     General: UnitName=°, UnitFlags=#x00000004
//     Dynamic: Acceleration=6120, Deceleration=6120, Jerk=115600
//     Velo: FastManual=200, Maximum=18000
//     OtherSettings: AllowMotionCmdToSlave=true
//     encoder EncType=1
//       EncPara: ScaleFactorNumerator=4.29153e-05
//     drive DrvType=5
//       Analog: VeloReferenz=20000, TorqueSetpointScale=10, ScaleFactorActTorque=0.1
//       TimeComp: TaskDelayCycles=1
//     controller CtrType=1
//       CtrPara: PriorControlFactor=1
//         PosDiffControl: Enable=false
//         Observer: BandWidth=20
//   AXIS Axis048_48 P1Ca_Ready2 (id 48) // P2备用2
//     General: UnitName=°, UnitFlags=#x00000004
//     Dynamic: Acceleration=24909.1, Deceleration=24909.1, Jerk=838463
//     Velo: SlowManual=20, FastManual=100, Maximum=18000
//     OtherSettings: AllowMotionCmdToSlave=true
//     encoder EncType=1
//       EncPara: ScaleFactorNumerator=4.29153e-05
//     drive DrvType=5
//       Analog: VeloReferenz=20000, TorqueSetpointScale=10, ScaleFactorActTorque=0.1
//       TimeComp: TaskDelayCycles=1
//     controller CtrType=1
//       CtrPara: PriorControlFactor=1
//         Observer: BandWidth=20
//   AXIS Axis049_1 P2M1_AnCarryingLine (id 49) // 1号叠台正极送片搬运平移
//     Dynamic: Acceleration=42600, Deceleration=42600, Jerk=1440290
//     Velo: FastManual=200, Maximum=3000
//     OtherSettings: AllowMotionCmdToSlave=true
//     encoder EncType=19
//       EncPara: MaxCount=#xffffffff
//     drive DrvType=16
//       DrvPara: MaxCount=#xffffffff, DriveControlDWord=#x00020100
//         Analog: VeloReferenz=3000, TorqueSetpointScale=10, ScaleFactorActTorque=0.1
//         TimeComp: TaskDelayCycles=1
//     controller CtrType=1
//       CtrPara: PriorControlFactor=1
//         Observer: BandWidth=20
//   AXIS Axis050_2 P2M1_AnCarryingUpDown (id 50) // 1号叠台正极送片搬运升降
//     Dynamic: Acceleration=79500, Deceleration=79500, Jerk=10712300
//     Velo: SlowManual=20, FastManual=100, Maximum=1000
//     OtherSettings: AllowMotionCmdToSlave=true
//     encoder EncType=19
//       EncPara: ScaleFactorNumerator=2.38419e-06, MaxCount=#xffffffff
//     drive DrvType=16
//       DrvPara: MaxCount=#xffffffff, DriveControlDWord=#x00020100
//         Analog: VeloReferenz=1000, TorqueSetpointScale=10, ScaleFactorActTorque=0.1
//         TimeComp: TaskDelayCycles=1
//     controller CtrType=1
//       CtrPara: PriorControlFactor=1
//         PosDiffControl: Enable=false
//         Observer: BandWidth=20
//   AXIS Axis051_3 P2M1_AnCarryingWhirling (id 51) // 1号叠台正极送片搬运旋转
//     General: UnitName=°
//     Dynamic: Acceleration=92400, Deceleration=92400, Jerk=1317560
//     Velo: FastManual=300, Maximum=12000
//     OtherSettings: AllowMotionCmdToSlave=true
//     encoder EncType=19
//       EncPara: ScaleFactorNumerator=2.86102e-05, ModuloFactor=114.59156, MaxCount=#xffffffff
//     drive DrvType=16
//       DrvPara: MaxCount=#xffffffff, DriveControlDWord=#x00020100
//         Analog: VeloReferenz=12000, TorqueSetpointScale=10, ScaleFactorActTorque=0.1
//         TimeComp: TaskDelayCycles=1
//     controller CtrType=1
//       CtrPara: PriorControlFactor=1
//         PosDiffControl: Enable=false
//         PID: PosKp=0
//         Observer: BandWidth=20
//   AXIS Axis052_4 P2M1_AnDTCarryingLine (id 52) // 1号叠台正极叠台搬运平移1
//     Dynamic: Acceleration=46200, Deceleration=46200, Jerk=1317560
//     Velo: SlowManual=20, FastManual=100, Maximum=3000
//     OtherSettings: AllowMotionCmdToSlave=true
//     encoder EncType=19
//       EncPara: MaxCount=#xffffffff
//     drive DrvType=16
//       DrvPara: MaxCount=#xffffffff, DriveControlDWord=#x00020100
//         Analog: VeloReferenz=3000, TorqueSetpointScale=10, ScaleFactorActTorque=0.1
//         TimeComp: TaskDelayCycles=1
//     controller CtrType=1
//       CtrPara: PriorControlFactor=1
//         Observer: BandWidth=20
//   AXIS Axis053_5 P2M1_AnDTCarryingUpDown (id 53) // 1号叠台正极叠台搬运升降
//     Dynamic: Acceleration=15700, Deceleration=15700, Jerk=432439
//     Velo: SlowManual=20, FastManual=100, Maximum=1000
//     OtherSettings: AllowMotionCmdToSlave=true
//     encoder EncType=19
//       EncPara: ScaleFactorNumerator=2.38419e-06, MaxCount=#xffffffff
//     drive DrvType=16
//       DrvPara: MaxCount=#xffffffff, DriveControlDWord=#x00020100
//         Analog: VeloReferenz=1000, TorqueSetpointScale=10, ScaleFactorActTorque=0.1
//         TimeComp: TaskDelayCycles=1
//     controller CtrType=1
//       CtrPara: PriorControlFactor=1
//         PosDiffControl: Enable=false
//         Observer: BandWidth=20
//   AXIS Axis054_6 P2M1_AndeviationX1 (id 54) // 1号叠台正极纠偏平台X1
//     Dynamic: Acceleration=11280, Deceleration=11280, Jerk=387922
//     Velo: SlowManual=10, FastManual=30, Maximum=800
//     OtherSettings: AllowMotionCmdToSlave=true
//     encoder EncType=19
//       EncPara: ScaleFactorNumerator=5.96046e-07, MaxCount=#xffffffff
//     drive DrvType=16
//       DrvPara: MaxCount=#xffffffff, DriveControlDWord=#x00020100
//         Analog: VeloReferenz=800, TorqueSetpointScale=10, ScaleFactorActTorque=0.1
//         TimeComp: TaskDelayCycles=1
//     controller CtrType=1
//       CtrPara: PriorControlFactor=1
//         Observer: BandWidth=20
//   AXIS Axis055_7 P2M1_AndeviationX2 (id 55) // 1号叠台正极纠偏平台X2
//     Dynamic: Acceleration=11440, Deceleration=11440, Jerk=380447
//     Velo: FastManual=300, Maximum=800
//     OtherSettings: AllowMotionCmdToSlave=true
//     encoder EncType=19
//       EncPara: ScaleFactorNumerator=5.96046e-07, ModuloFactor=114.59156, MaxCount=#xffffffff
//     drive DrvType=16
//       DrvPara: MaxCount=#xffffffff, DriveControlDWord=#x00020100
//         Analog: VeloReferenz=800, TorqueSetpointScale=10, ScaleFactorActTorque=0.1
//         TimeComp: TaskDelayCycles=1
//     controller CtrType=1
//       CtrPara: PriorControlFactor=1
//         PID: PosKp=0
//         Observer: BandWidth=20
//   AXIS Axis056_8 P2M1_AndeviationY (id 56) // 1号叠台正极纠偏平台Y
//     Dynamic: Acceleration=11360, Deceleration=11360, Jerk=384076
//     Velo: SlowManual=20, FastManual=100, Maximum=800
//     OtherSettings: AllowMotionCmdToSlave=true
//     encoder EncType=19
//       EncPara: ScaleFactorNumerator=5.96046e-07, MaxCount=#xffffffff
//     drive DrvType=16
//       DrvPara: MaxCount=#xffffffff, DriveControlDWord=#x00020100
//         Analog: VeloReferenz=800, TorqueSetpointScale=10, ScaleFactorActTorque=0.1
//         TimeComp: TaskDelayCycles=1
//     controller CtrType=1
//       CtrPara: PriorControlFactor=1
//         Observer: BandWidth=20
//   AXIS Axis057_9 P2M1_CaCarryingLine1 (id 57) // 1号叠台负极送片搬运1平移
//     Dynamic: Acceleration=34109.1, Deceleration=34109.1, Jerk=1222090
//     Velo: SlowManual=20, FastManual=100, Maximum=3000
//     OtherSettings: AllowMotionCmdToSlave=true
//     encoder EncType=19
//       EncPara: MaxCount=#xffffffff
//     drive DrvType=16
//       DrvPara: MaxCount=#xffffffff, DriveControlDWord=#x00020100
//         Analog: VeloReferenz=3000, TorqueSetpointScale=10, ScaleFactorActTorque=0.1
//         TimeComp: TaskDelayCycles=1
//     controller CtrType=1
//       CtrPara: PriorControlFactor=1
//         Observer: BandWidth=20
//   AXIS Axis058_10 P2M1_CaCarryingUpDown1 (id 58) // 1号叠台负极送片搬运1升降
//     Dynamic: Acceleration=33750, Deceleration=33750, Jerk=3254470
//     Velo: SlowManual=10, FastManual=30, Maximum=1000
//     OtherSettings: AllowMotionCmdToSlave=true
//     encoder EncType=19
//       EncPara: ScaleFactorNumerator=2.38419e-06, MaxCount=#xffffffff
//     drive DrvType=16
//       DrvPara: MaxCount=#xffffffff, DriveControlDWord=#x00020100
//         Analog: VeloReferenz=1000, TorqueSetpointScale=10, ScaleFactorActTorque=0.1
//         TimeComp: TaskDelayCycles=1
//     controller CtrType=1
//       CtrPara: PriorControlFactor=1
//         PosDiffControl: Enable=false
//         Observer: BandWidth=20
//   AXIS Axis059_11 P2M1_CaCarryingWhirling1 (id 59) // 1号叠台负极送片搬运1旋转
//     General: UnitName=°
//     Dynamic: Acceleration=190800, Deceleration=190800, Jerk=5141900
//     Velo: Maximum=12000
//     OtherSettings: AllowMotionCmdToSlave=true
//     encoder EncType=19
//       EncPara: ScaleFactorNumerator=2.86102e-05, MaxCount=#xffffffff
//     drive DrvType=16
//       DrvPara: MaxCount=#xffffffff, DriveControlDWord=#x00020100
//         Analog: VeloReferenz=12000, TorqueSetpointScale=10, ScaleFactorActTorque=0.1
//         TimeComp: TaskDelayCycles=1
//     controller CtrType=1
//       CtrPara: PriorControlFactor=1
//         PosDiffControl: Enable=false
//         Observer: BandWidth=20
//   AXIS Axis060_12 P2M1_CaCarryingLine2 (id 60) // 1号叠台负极送片搬运2平移
//     Dynamic: Acceleration=46500, Deceleration=46500, Jerk=1310450
//     Velo: Maximum=3000
//     OtherSettings: AllowMotionCmdToSlave=true
//     encoder EncType=19
//       EncPara: MaxCount=#xffffffff
//     drive DrvType=16
//       DrvPara: MaxCount=#xffffffff, DriveControlDWord=#x00020100
//         Analog: VeloReferenz=3000, TorqueSetpointScale=10, ScaleFactorActTorque=0.1
//         TimeComp: TaskDelayCycles=1
//     controller CtrType=1
//       CtrPara: PriorControlFactor=1
//         Observer: BandWidth=20
//   AXIS Axis061_13 P2M1_CaCarryingUpDown2 (id 61) // 1号叠台负极送片搬运2升降
//     Dynamic: Acceleration=25000, Deceleration=25000, Jerk=1250000
//     Velo: Maximum=1000
//     OtherSettings: AllowMotionCmdToSlave=true
//     encoder EncType=19
//       EncPara: ScaleFactorNumerator=2.38419e-06, MaxCount=#xffffffff
//     drive DrvType=16
//       DrvPara: MaxCount=#xffffffff, DriveControlDWord=#x00020100
//         Analog: VeloReferenz=1000, TorqueSetpointScale=10, ScaleFactorActTorque=0.1
//         TimeComp: TaskDelayCycles=1
//     controller CtrType=1
//       CtrPara: PriorControlFactor=1
//         PosDiffControl: Enable=false
//         Observer: BandWidth=20
//   AXIS Axis062_14 P2M1_CaBelt (id 62) // 1号叠台负极送片皮带
//     Dynamic: Acceleration=41919, Deceleration=41919, Jerk=1154610
//     Velo: Maximum=2670
//     OtherSettings: AllowMotionCmdToSlave=true
//     encoder EncType=19
//       EncPara: ScaleFactorNumerator=6.36662e-06, MaxCount=#xffffffff
//     drive DrvType=16
//       DrvPara: MaxCount=#xffffffff, DriveControlDWord=#x00020100
//         Analog: VeloReferenz=2670, TorqueSetpointScale=10, ScaleFactorActTorque=0.1
//         TimeComp: TaskDelayCycles=1
//     controller CtrType=1
//       CtrPara: PriorControlFactor=1
//         PosDiffControl: Enable=false
//         Observer: BandWidth=20
//   AXIS Axis063_15 P2M1_CaDTCarryingLine (id 63) // 1号叠台负极叠台搬运平移
//     Dynamic: Acceleration=46500, Deceleration=46500, Jerk=1310450
//     Velo: Maximum=3000
//     OtherSettings: AllowMotionCmdToSlave=true
//     encoder EncType=19
//       EncPara: MaxCount=#xffffffff
//     drive DrvType=16
//       DrvPara: MaxCount=#xffffffff, DriveControlDWord=#x00020100
//         Analog: VeloReferenz=3000, TorqueSetpointScale=10, ScaleFactorActTorque=0.1
//         TimeComp: TaskDelayCycles=1
//     controller CtrType=1
//       CtrPara: PriorControlFactor=1
//         Observer: BandWidth=20
//   AXIS Axis064_16 P2M1_CaDTCarryingUpDown (id 64) // 1号叠台负极叠台搬运升降
//     Dynamic: Acceleration=15800, Deceleration=15800, Jerk=430414
//     Velo: Maximum=1000
//     OtherSettings: AllowMotionCmdToSlave=true
//     encoder EncType=19
//       EncPara: ScaleFactorNumerator=2.38419e-06, MaxCount=#xffffffff
//     drive DrvType=16
//       DrvPara: MaxCount=#xffffffff, DriveControlDWord=#x00020100
//         Analog: VeloReferenz=1000, TorqueSetpointScale=10, ScaleFactorActTorque=0.1
//         TimeComp: TaskDelayCycles=1
//     controller CtrType=1
//       CtrPara: PriorControlFactor=1
//         PosDiffControl: Enable=false
//         Observer: BandWidth=20
//   AXIS Axis065_17 P2M1_CadeviationX1 (id 65) // 1号叠台负极纠偏平台X1
//     Dynamic: Acceleration=11440, Deceleration=11440, Jerk=380447
//     Velo: FastManual=200, Maximum=800
//     OtherSettings: AllowMotionCmdToSlave=true
//     encoder EncType=19
//       EncPara: ScaleFactorNumerator=5.96046e-07, MaxCount=#xffffffff
//     drive DrvType=16
//       DrvPara: MaxCount=#xffffffff, DriveControlDWord=#x00020100
//         Analog: VeloReferenz=800, TorqueSetpointScale=10, ScaleFactorActTorque=0.1
//         TimeComp: TaskDelayCycles=1
//     controller CtrType=1
//       CtrPara: PriorControlFactor=1
//         Observer: BandWidth=20
//   AXIS Axis066_18 P2M1_CadeviationX2 (id 66) // 1号叠台负极纠偏平台X2
//     Dynamic: Acceleration=11360, Deceleration=11360, Jerk=384076
//     Velo: FastManual=200, Maximum=800
//     OtherSettings: AllowMotionCmdToSlave=true
//     encoder EncType=19
//       EncPara: ScaleFactorNumerator=5.96046e-07, MaxCount=#xffffffff
//     drive DrvType=16
//       DrvPara: MaxCount=#xffffffff, DriveControlDWord=#x00020100
//         Analog: VeloReferenz=800, TorqueSetpointScale=10, ScaleFactorActTorque=0.1
//         TimeComp: TaskDelayCycles=1
//     controller CtrType=1
//       CtrPara: PriorControlFactor=1
//         Observer: BandWidth=20
//   AXIS Axis067_19 P2M1_CadeviationY (id 67) // 1号叠台负极纠偏平台Y
//     Dynamic: Acceleration=11120, Deceleration=11120, Jerk=396328
//     Velo: FastManual=200, Maximum=800
//     OtherSettings: AllowMotionCmdToSlave=true
//     encoder EncType=19
//       EncPara: ScaleFactorNumerator=5.96046e-07, MaxCount=#xffffffff
//     drive DrvType=16
//       DrvPara: MaxCount=#xffffffff, DriveControlDWord=#x00020100
//         Analog: VeloReferenz=800, TorqueSetpointScale=10, ScaleFactorActTorque=0.1
//         TimeComp: TaskDelayCycles=1
//     controller CtrType=1
//       CtrPara: PriorControlFactor=1
//         Observer: BandWidth=20
//   AXIS Axis068_20 P2M1_SEPTAunwinding (id 68) // 1号叠台隔膜放卷
//     General: UnitName=°
//     Dynamic: Acceleration=4932, Deceleration=4932, Jerk=91308.6
//     Velo: SlowManual=50, FastManual=100, Maximum=3600
//     OtherSettings: AllowMotionCmdToSlave=true
//     encoder EncType=19
//       EncPara: ScaleFactorNumerator=8.58307e-06, MaxCount=#xffffffff
//     drive DrvType=16
//       DrvPara: MaxCount=#xffffffff, DriveControlDWord=#x00020100
//         Analog: VeloReferenz=3600, TorqueSetpointScale=10, ScaleFactorActTorque=0.1
//         TimeComp: TaskDelayCycles=1
//     controller CtrType=1
//       CtrPara: PriorControlFactor=1
//         PosDiffControl: Enable=false, Range=10
//         Observer: BandWidth=20
//   AXIS Axis069_21 P2M1_SEPTAdeviation1 (id 69) // 1号叠台隔膜放卷纠偏
//     Dynamic: Acceleration=3060, Deceleration=3060, Jerk=88335.8
//     Velo: SlowManual=50, FastManual=100, Maximum=200
//     OtherSettings: AllowMotionCmdToSlave=true
//     encoder EncType=19
//       EncPara: ScaleFactorNumerator=4.76837e-07, MaxCount=#xffffffff
//     drive DrvType=16
//       DrvPara: MaxCount=#xffffffff, DriveControlDWord=#x00020100
//         Analog: VeloReferenz=200, TorqueSetpointScale=10, ScaleFactorActTorque=0.1
//         TimeComp: TaskDelayCycles=1
//     controller CtrType=1
//       CtrPara: PriorControlFactor=1
//         PosDiffControl: Range=10
//         Observer: BandWidth=20
//   AXIS Axis070_22 P2M1_SEPTAdeviation2 (id 70) // 1号叠台隔膜尾部纠偏
//     Dynamic: Acceleration=3850, Deceleration=3850, Jerk=109796
//     Velo: Maximum=250
//     OtherSettings: AllowMotionCmdToSlave=true
//     encoder EncType=19
//       EncPara: ScaleFactorNumerator=5.96046e-07, MaxCount=#xffffffff
//     drive DrvType=16
//       DrvPara: MaxCount=#xffffffff, DriveControlDWord=#x00020100
//         Analog: VeloReferenz=250, TorqueSetpointScale=10, ScaleFactorActTorque=0.1
//         TimeComp: TaskDelayCycles=1
//     controller CtrType=1
//       CtrPara: PriorControlFactor=1
//         Observer: BandWidth=20
//   AXIS Axis071_23 P2M1_SEPTATension (id 71) // 1号叠台隔膜摆杆张力
//     General: UnitName=°
//     Dynamic: Acceleration=62400, Deceleration=62400, Jerk=1738290
//     Velo: Maximum=4000
//     OtherSettings: AllowMotionCmdToSlave=true
//     encoder EncType=19
//       EncPara: ScaleFactorNumerator=4.29153e-05, Offset=-19.1455882125, MaxCount=#xffffffff, ReferenceSystem=1
//     drive DrvType=16
//       DrvPara: MaxCount=#xffffffff, DriveControlDWord=#x00020000
//         Analog: VeloReferenz=18000, TorqueSetpointScale=10, ScaleFactorActTorque=0.1
//         TimeComp: TaskDelayCycles=1
//     controller CtrType=1
//       CtrPara: PriorControlFactor=1
//         PosDiffControl: Enable=false
//         Observer: BandWidth=20
//   AXIS Axis072_24 P2M1_SEPTATCache (id 72) // 1号叠台隔膜缓存
//     Dynamic: Acceleration=46500, Deceleration=46500, Jerk=1310450
//     Velo: Maximum=3000
//     OtherSettings: AllowMotionCmdToSlave=true
//     encoder EncType=19
//       EncPara: MaxCount=#xffffffff
//     drive DrvType=16
//       DrvPara: MaxCount=#xffffffff, DriveControlDWord=#x00020100
//         Analog: VeloReferenz=3000, TorqueSetpointScale=10, ScaleFactorActTorque=0.1
//         TimeComp: TaskDelayCycles=1
//     controller CtrType=1
//       CtrPara: PriorControlFactor=1
//         Observer: BandWidth=20
//   AXIS Axis073_25 P2M1_SEPTATLine (id 73) // 1号叠台隔膜平移
//     Dynamic: Acceleration=46800, Deceleration=46800, Jerk=1303710
//     Velo: Maximum=3000
//     OtherSettings: AllowMotionCmdToSlave=true
//     encoder EncType=19
//       EncPara: MaxCount=#xffffffff
//     drive DrvType=16
//       DrvPara: MaxCount=#xffffffff, DriveControlDWord=#x00020100
//         Analog: VeloReferenz=3000, TorqueSetpointScale=10, ScaleFactorActTorque=0.1
//         TimeComp: TaskDelayCycles=1
//     controller CtrType=1
//       CtrPara: PriorControlFactor=1
//         Observer: BandWidth=20
//   AXIS Axis074_26 P2M1_DTUpDown (id 74) // 1号叠台叠台升降
//     Dynamic: Acceleration=7800, Deceleration=7800, Jerk=217286
//     Velo: Maximum=500
//     OtherSettings: AllowMotionCmdToSlave=true
//     encoder EncType=19
//       EncPara: ScaleFactorNumerator=5.96046e-07, MaxCount=#xffffffff
//     drive DrvType=16
//       DrvPara: MaxCount=#xffffffff, DriveControlDWord=#x00020100
//         Analog: VeloReferenz=250, TorqueSetpointScale=10, ScaleFactorActTorque=0.1
//         TimeComp: TaskDelayCycles=1
//     controller CtrType=1
//       CtrPara: PriorControlFactor=1
//         PosDiffControl: Enable=false
//         Observer: BandWidth=20
//   AXIS Axis075_27 P2M1_LeftYDLine (id 75) // 1号叠台左压刀开合
//     Dynamic: Acceleration=31400, Deceleration=31400, Jerk=864877
//     OtherSettings: AllowMotionCmdToSlave=true
//     encoder EncType=19
//       EncPara: ScaleFactorNumerator=1.3113e-05, MaxCount=#xffffffff
//     drive DrvType=16
//       DrvPara: MaxCount=#xffffffff, DriveControlDWord=#x00020100
//         Analog: VeloReferenz=5500, TorqueSetpointScale=10, ScaleFactorActTorque=0.1
//         TimeComp: TaskDelayCycles=1
//     controller CtrType=1
//       CtrPara: PriorControlFactor=1
//         PosDiffControl: Enable=false
//         Observer: BandWidth=20
//   AXIS Axis076_28 P2M1_LeftYDUpDown (id 76) // 1号叠台左压刀升降
//     Dynamic: Acceleration=4075.47, Deceleration=4075.47, Jerk=110730
//     Velo: Maximum=250
//     OtherSettings: AllowMotionCmdToSlave=true
//     encoder EncType=19
//       EncPara: ScaleFactorNumerator=5.96046e-07, MaxCount=#xffffffff
//     drive DrvType=16
//       DrvPara: MaxCount=#xffffffff, DriveControlDWord=#x00020100
//         Analog: VeloReferenz=250, TorqueSetpointScale=10, ScaleFactorActTorque=0.1
//         TimeComp: TaskDelayCycles=1
//     controller CtrType=1
//       CtrPara: PriorControlFactor=1
//         PosDiffControl: Enable=false
//         Observer: BandWidth=20
//   AXIS Axis077_29 P2M1_RightYDLine (id 77) // 1号叠台右压刀开合
//     Dynamic: Acceleration=31400, Deceleration=31400, Jerk=864877
//     OtherSettings: AllowMotionCmdToSlave=true
//     encoder EncType=19
//       EncPara: ScaleFactorNumerator=1.3113e-05, Offset=0.02799504156, MaxCount=#xffffffff
//     drive DrvType=16
//       DrvPara: MaxCount=#xffffffff, DriveControlDWord=#x00020100
//         Analog: VeloReferenz=5500, TorqueSetpointScale=10, ScaleFactorActTorque=0.1
//         TimeComp: TaskDelayCycles=1
//     controller CtrType=1
//       CtrPara: PriorControlFactor=1
//         PosDiffControl: Enable=false
//         Observer: BandWidth=20
//   AXIS Axis078_30 P2M1_RightYDUpDown (id 78) // 1号叠台右压刀升降
//     Dynamic: Acceleration=4000, Deceleration=4000, Jerk=106667
//     Velo: Maximum=250
//     OtherSettings: AllowMotionCmdToSlave=true
//     encoder EncType=19
//       EncPara: ScaleFactorNumerator=5.96046e-07, MaxCount=#xffffffff
//     drive DrvType=16
//       DrvPara: MaxCount=#xffffffff, DriveControlDWord=#x00020100
//         Analog: VeloReferenz=250, TorqueSetpointScale=10, ScaleFactorActTorque=0.1
//         TimeComp: TaskDelayCycles=1
//     controller CtrType=1
//       CtrPara: PriorControlFactor=1
//         PosDiffControl: Enable=false
//         Observer: BandWidth=20
//   AXIS Axis079_31 P2M1_TailCurlLine (id 79) // 1号叠台尾卷夹电芯平移
//     Dynamic: Acceleration=1773, Deceleration=1773, Jerk=18880.1
//     Velo: Maximum=720
//     OtherSettings: AllowMotionCmdToSlave=true
//     encoder EncType=19
//       EncPara: ScaleFactorNumerator=1.72191e-06, Offset=57.90649177236, MaxCount=#xffffffff
//     drive DrvType=16
//       DrvPara: MaxCount=#xffffffff, DriveControlDWord=#x00020100
//         Analog: VeloReferenz=720, TorqueSetpointScale=10, ScaleFactorActTorque=0.1
//         TimeComp: TaskDelayCycles=1
//     controller CtrType=1
//       CtrPara: PriorControlFactor=1
//         PosDiffControl: Enable=false
//         Observer: BandWidth=20
//   AXIS Axis080_32 P2M1_TailCurlUpDown (id 80) // 1号叠台尾卷夹电芯升降
//     Dynamic: Acceleration=4210, Deceleration=4210, Jerk=103650
//     Velo: Maximum=250
//     OtherSettings: AllowMotionCmdToSlave=true
//     encoder EncType=19
//       EncPara: ScaleFactorNumerator=5.96046e-07, Offset=168.26270241552, MaxCount=#xffffffff, ReferenceSystem=1
//     drive DrvType=16
//       DrvPara: MaxCount=#xffffffff, DriveControlDWord=#x00020100
//         Analog: VeloReferenz=250, TorqueSetpointScale=10, ScaleFactorActTorque=0.1
//         TimeComp: TaskDelayCycles=1
//     controller CtrType=1
//       CtrPara: PriorControlFactor=1
//         PosDiffControl: Enable=false
//         Observer: BandWidth=20
//   AXIS Axis081_33 P2M1_TailCurlRetracting (id 81) // 1号叠台尾卷夹电芯伸缩
//     Dynamic: Acceleration=24444.4, Deceleration=24444.4, Jerk=1344440
//     OtherSettings: AllowMotionCmdToSlave=true
//     encoder EncType=19
//       EncPara: ScaleFactorNumerator=1.07288e-05, MaxCount=#xffffffff
//     drive DrvType=16
//       DrvPara: MaxCount=#xffffffff, DriveControlDWord=#x00020100
//         Analog: VeloReferenz=4500, TorqueSetpointScale=10, ScaleFactorActTorque=0.1
//         TimeComp: TaskDelayCycles=1
//     controller CtrType=1
//       CtrPara: PriorControlFactor=1
//         PosDiffControl: Enable=false
//         Observer: BandWidth=20
//   AXIS Axis082_34 P2M1_TailCurlWhirling (id 82) // 1号叠台尾卷夹电芯旋转
//     General: UnitName=°
//     Dynamic: Acceleration=13600, Deceleration=13600, Jerk=256889
//     Velo: Maximum=900
//     OtherSettings: AllowMotionCmdToSlave=true
//     encoder EncType=19
//       EncPara: ScaleFactorNumerator=2.14577e-06, MaxCount=#xffffffff, ReferenceSystem=1
//     drive DrvType=16
//       DrvPara: MaxCount=#xffffffff, DriveControlDWord=#x00020100
//         Analog: VeloReferenz=900, TorqueSetpointScale=10, ScaleFactorActTorque=0.1
//         TimeComp: TaskDelayCycles=1
//     controller CtrType=1
//       CtrPara: PriorControlFactor=1
//         PosDiffControl: Enable=false
//         Observer: BandWidth=20
//   AXIS Axis083_35 P2M1_TailCurlSEPTALine (id 83) // 1号叠台夹膜平移
//     Dynamic: Acceleration=7875.72, Deceleration=7875.72, Jerk=148532
//     Velo: Maximum=720
//     OtherSettings: AllowMotionCmdToSlave=true
//     encoder EncType=19
//       EncPara: ScaleFactorNumerator=1.72191e-06, Offset=-4.132584e-05, MaxCount=#xffffffff, ReferenceSystem=1
//     drive DrvType=16
//       DrvPara: MaxCount=#xffffffff, DriveControlDWord=#x00020100
//         Analog: VeloReferenz=720, TorqueSetpointScale=10, ScaleFactorActTorque=0.1
//         TimeComp: TaskDelayCycles=1
//     controller CtrType=1
//       CtrPara: PriorControlFactor=1
//         PosDiffControl: Enable=false
//         Observer: BandWidth=20
//   AXIS Axis084_36 P2M1_TailCurlSEPTAUpDown (id 84) // 1号叠台夹膜升降
//     Dynamic: Acceleration=3950, Deceleration=3950, Jerk=107603
//     Velo: Maximum=250
//     OtherSettings: AllowMotionCmdToSlave=true
//     encoder EncType=19
//       EncPara: ScaleFactorNumerator=5.96046e-07, MaxCount=#xffffffff
//     drive DrvType=16
//       DrvPara: MaxCount=#xffffffff, DriveControlDWord=#x00020100
//         Analog: VeloReferenz=250, TorqueSetpointScale=10, ScaleFactorActTorque=0.1
//         TimeComp: TaskDelayCycles=1
//     controller CtrType=1
//       CtrPara: PriorControlFactor=1
//         PosDiffControl: Enable=false
//         Observer: BandWidth=20
//   AXIS Axis085_37 P2M1_LCurlingneedleLine (id 85) // 1号叠台长卷针平移
//     Dynamic: Acceleration=20410, Deceleration=20410, Jerk=562170
//     Velo: Maximum=1300
//     OtherSettings: AllowMotionCmdToSlave=true
//     encoder EncType=19
//       EncPara: ScaleFactorNumerator=0.01, MaxCount=#xffffffff
//     drive DrvType=16
//       DrvPara: MaxCount=#xffffffff, DriveControlDWord=#x00020000
//         Analog: VeloReferenz=1300, TorqueSetpointScale=10, ScaleFactorActTorque=0.1
//         TimeComp: TaskDelayCycles=1
//     controller CtrType=1
//       CtrPara: PriorControlFactor=1
//         PosDiffControl: Enable=false
//         Observer: BandWidth=20
//   AXIS Axis086_38 P2M1_SCurlingneedleLine (id 86) // 1号叠台短卷针平移
//     Dynamic: Acceleration=20020, Deceleration=20020, Jerk=570941
//     Velo: Maximum=1300
//     OtherSettings: AllowMotionCmdToSlave=true
//     encoder EncType=19
//       EncPara: ScaleFactorNumerator=0.01, MaxCount=#xffffffff
//     drive DrvType=16
//       DrvPara: MaxCount=#xffffffff, DriveControlDWord=#x00020000
//         Analog: VeloReferenz=1300, TorqueSetpointScale=10, ScaleFactorActTorque=0.1
//         TimeComp: TaskDelayCycles=1
//     controller CtrType=1
//       CtrPara: PriorControlFactor=1
//         PosDiffControl: Enable=false
//         Observer: BandWidth=20
//   AXIS Axis087_39 P2M1_LCurlingneedleWhirling (id 87) // 1号叠台长卷针旋转
//     General: UnitName=°, UnitFlags=#x00000004
//     Dynamic: Acceleration=37440, Deceleration=37440, Jerk=1042970
//     Velo: Maximum=2400
//     OtherSettings: AllowMotionCmdToSlave=true
//     encoder EncType=19
//       EncPara: ScaleFactorNumerator=0.018, MaxCount=#xffffffff
//     drive DrvType=16
//       DrvPara: MaxCount=#xffffffff, DriveControlDWord=#x00020000
//         Analog: VeloReferenz=2400, TorqueSetpointScale=10, ScaleFactorActTorque=0.1
//         TimeComp: TaskDelayCycles=1
//     controller CtrType=1
//       CtrPara: PriorControlFactor=1
//         PosDiffControl: Enable=false
//         Observer: BandWidth=20
//   AXIS Axis088_40 P2M1_SCurlingneedleWhirling (id 88) // 1号叠台短卷针旋转
//     General: UnitName=°, UnitFlags=#x00000004
//     Dynamic: Acceleration=37680, Deceleration=37680, Jerk=1037850
//     Velo: Maximum=2400
//     OtherSettings: AllowMotionCmdToSlave=true
//     encoder EncType=19
//       EncPara: ScaleFactorNumerator=0.018, MaxCount=#xffffffff
//     drive DrvType=16
//       DrvPara: MaxCount=#xffffffff, DriveControlDWord=#x00020000
//         Analog: VeloReferenz=2400, TorqueSetpointScale=10, ScaleFactorActTorque=0.1
//         TimeComp: TaskDelayCycles=1
//     controller CtrType=1
//       CtrPara: PriorControlFactor=1
//         PosDiffControl: Enable=false
//         Observer: BandWidth=20
//   AXIS Axis089_41 P2M1_GluingLine (id 89) // 1号叠台侧贴夹平移
//     Dynamic: Acceleration=775, Deceleration=775, Jerk=2184.09
//     Velo: Maximum=500
//     OtherSettings: AllowMotionCmdToSlave=true
//     encoder EncType=19
//       EncPara: ScaleFactorNumerator=1.19209e-06, MaxCount=#xffffffff
//     drive DrvType=16
//       DrvPara: MaxCount=#xffffffff, DriveControlDWord=#x00020100
//         Analog: VeloReferenz=500, TorqueSetpointScale=10, ScaleFactorActTorque=0.1
//         TimeComp: TaskDelayCycles=1
//     controller CtrType=1
//       CtrPara: PriorControlFactor=1
//         PosDiffControl: Enable=false
//         Observer: BandWidth=20
//   AXIS Axis090_42 P2M1_GluingWhirling (id 90) // 1号叠台侧贴夹旋转
//     General: UnitName=°
//     Dynamic: Acceleration=1413, Deceleration=1413, Jerk=3891.95
//     Velo: Maximum=900
//     OtherSettings: AllowMotionCmdToSlave=true
//     encoder EncType=19
//       EncPara: ScaleFactorNumerator=2.14577e-06, MaxCount=#xffffffff
//     drive DrvType=16
//       DrvPara: MaxCount=#xffffffff, DriveControlDWord=#x00020100
//         Analog: VeloReferenz=900, TorqueSetpointScale=10, ScaleFactorActTorque=0.1
//         TimeComp: TaskDelayCycles=1
//     controller CtrType=1
//       CtrPara: PriorControlFactor=1
//         PosDiffControl: Enable=false
//         Observer: BandWidth=20
//   AXIS Axis091_43 P2M1_GluingRetracting (id 91) // 1号叠台贴胶头进退
//     Dynamic: Acceleration=15500, Deceleration=15500, Jerk=436818
//     Velo: Maximum=1000
//     OtherSettings: AllowMotionCmdToSlave=true
//     encoder EncType=19
//       EncPara: ScaleFactorNumerator=2.38419e-06, MaxCount=#xffffffff
//     drive DrvType=16
//       DrvPara: MaxCount=#xffffffff, DriveControlDWord=#x00020100
//         Analog: VeloReferenz=1000, TorqueSetpointScale=10, ScaleFactorActTorque=0.1
//         TimeComp: TaskDelayCycles=1
//     controller CtrType=1
//       CtrPara: PriorControlFactor=1
//         PosDiffControl: Enable=false
//         Observer: BandWidth=20
//   AXIS Axis092_44 P2M1_GluingUpDown (id 92) // 1号叠台拉胶升降
//     Dynamic: Acceleration=775, Deceleration=775, Jerk=2184.09
//     Velo: Maximum=500
//     OtherSettings: AllowMotionCmdToSlave=true
//     encoder EncType=19
//       EncPara: ScaleFactorNumerator=1.19209e-06, MaxCount=#xffffffff
//     drive DrvType=16
//       DrvPara: MaxCount=#xffffffff, DriveControlDWord=#x00020100
//         Analog: VeloReferenz=500, TorqueSetpointScale=10, ScaleFactorActTorque=0.1
//         TimeComp: TaskDelayCycles=1
//     controller CtrType=1
//       CtrPara: PriorControlFactor=1
//         PosDiffControl: Enable=false
//         Observer: BandWidth=20
//   AXIS Axis093_45 P2M1_Standby1 (id 93) // 1号叠台叠片备用2
//     Dynamic: Acceleration=30000, Deceleration=30000, Jerk=900000
//     OtherSettings: AllowMotionCmdToSlave=true
//     encoder EncType=1
//     drive DrvType=5
//       Analog: TorqueSetpointScale=10, ScaleFactorActTorque=0.1
//       TimeComp: TaskDelayCycles=1
//     controller CtrType=1
//       CtrPara: PriorControlFactor=1
//         Observer: BandWidth=20
//   AXIS Axis094_46 P2M1_Standby2 (id 94) // 1号叠台叠片备用2
//     OtherSettings: AllowMotionCmdToSlave=true
//     encoder EncType=1
//     drive DrvType=5
//       Analog: TorqueSetpointScale=10, ScaleFactorActTorque=0.1
//       TimeComp: TaskDelayCycles=1
//     controller CtrType=1
//       CtrPara: PriorControlFactor=1
//         Observer: BandWidth=20
//   AXIS Axis095_47 P2M2_AnCarryingLine (id 95) // 2号叠片正极送片搬运平移
//     Dynamic: Acceleration=45900, Deceleration=45900, Jerk=1325040
//     Velo: Maximum=3000
//     OtherSettings: AllowMotionCmdToSlave=true
//     encoder EncType=19
//       EncPara: MaxCount=#xffffffff
//     drive DrvType=16
//       DrvPara: MaxCount=#xffffffff, DriveControlDWord=#x00020100
//         Analog: VeloReferenz=3000, TorqueSetpointScale=10, ScaleFactorActTorque=0.1
//         TimeComp: TaskDelayCycles=1
//     controller CtrType=1
//       CtrPara: PriorControlFactor=1
//         Observer: BandWidth=20
//   AXIS Axis096_48 P2M2_AnCarryingUpDown (id 96) // 2号正极送片搬运升降
//     Dynamic: Acceleration=79000, Deceleration=79000, Jerk=10760300
//     Velo: Maximum=1000
//     OtherSettings: AllowMotionCmdToSlave=true
//     encoder EncType=19
//       EncPara: ScaleFactorNumerator=2.38419e-06, MaxCount=#xffffffff
//     drive DrvType=16
//       DrvPara: MaxCount=#xffffffff, DriveControlDWord=#x00020100
//         Analog: VeloReferenz=1000, TorqueSetpointScale=10, ScaleFactorActTorque=0.1
//         TimeComp: TaskDelayCycles=1
//     controller CtrType=1
//       CtrPara: PriorControlFactor=1
//         PosDiffControl: Enable=false
//         Observer: BandWidth=20
//   AXIS Axis097_49 P2M2_AnCarryingWhirling (id 97) // 2号正极送片搬运旋转
//     General: UnitName=°
//     Dynamic: Acceleration=189600, Deceleration=189600, Jerk=5164970
//     Velo: Maximum=12000
//     OtherSettings: AllowMotionCmdToSlave=true
//     encoder EncType=19
//       EncPara: ScaleFactorNumerator=2.86102e-05, MaxCount=#xffffffff
//     drive DrvType=16
//       DrvPara: MaxCount=#xffffffff, DriveControlDWord=#x00020100
//         Analog: VeloReferenz=12000, TorqueSetpointScale=10, ScaleFactorActTorque=0.1
//         TimeComp: TaskDelayCycles=1
//     controller CtrType=1
//       CtrPara: PriorControlFactor=1
//         PosDiffControl: Enable=false
//         Observer: BandWidth=20
//   AXIS Axis098_50 P2M2_AnDTCarryingLine (id 98) // 2号正极叠台搬运平移
//     Dynamic: Acceleration=48000, Deceleration=48000, Jerk=1280000
//     Velo: Maximum=3000
//     OtherSettings: AllowMotionCmdToSlave=true
//     encoder EncType=19
//       EncPara: MaxCount=#xffffffff
//     drive DrvType=16
//       DrvPara: MaxCount=#xffffffff, DriveControlDWord=#x00020100
//         Analog: VeloReferenz=3000, TorqueSetpointScale=10, ScaleFactorActTorque=0.1
//         TimeComp: TaskDelayCycles=1
//     controller CtrType=1
//       CtrPara: PriorControlFactor=1
//         Observer: BandWidth=20
//   AXIS Axis099_51 P2M2_AnDTCarryingUpDown (id 99) // 2号叠片正极搬运平移
//     Dynamic: Acceleration=15600, Deceleration=15600, Jerk=434571
//     Velo: Maximum=1000
//     OtherSettings: AllowMotionCmdToSlave=true
//     encoder EncType=19
//       EncPara: ScaleFactorNumerator=2.38419e-06, MaxCount=#xffffffff
//     drive DrvType=16
//       DrvPara: MaxCount=#xffffffff, DriveControlDWord=#x00020100
//         Analog: VeloReferenz=1000, TorqueSetpointScale=10, ScaleFactorActTorque=0.1
//         TimeComp: TaskDelayCycles=1
//     controller CtrType=1
//       CtrPara: PriorControlFactor=1
//         PosDiffControl: Enable=false
//         Observer: BandWidth=20
//   AXIS Axis100_52 P2M2_AndeviationX1 (id 100) // 2号叠片正极纠偏平台X1
//     Dynamic: Acceleration=11360, Deceleration=11360, Jerk=384076
//     Velo: Maximum=800
//     OtherSettings: AllowMotionCmdToSlave=true
//     encoder EncType=19
//       EncPara: ScaleFactorNumerator=5.96046e-07, MaxCount=#xffffffff
//     drive DrvType=16
//       DrvPara: MaxCount=#xffffffff, DriveControlDWord=#x00020100
//         Analog: VeloReferenz=800, TorqueSetpointScale=10, ScaleFactorActTorque=0.1
//         TimeComp: TaskDelayCycles=1
//     controller CtrType=1
//       CtrPara: PriorControlFactor=1
//         Observer: BandWidth=20
//   AXIS Axis101_53 P2M2_AndeviationX2 (id 101) // 2号叠片正极纠偏平台X2
//     Dynamic: Acceleration=11360, Deceleration=11360, Jerk=384076
//     Velo: Maximum=800
//     OtherSettings: AllowMotionCmdToSlave=true
//     encoder EncType=19
//       EncPara: ScaleFactorNumerator=5.96046e-07, MaxCount=#xffffffff
//     drive DrvType=16
//       DrvPara: MaxCount=#xffffffff, DriveControlDWord=#x00020100
//         Analog: VeloReferenz=800, TorqueSetpointScale=10, ScaleFactorActTorque=0.1
//         TimeComp: TaskDelayCycles=1
//     controller CtrType=1
//       CtrPara: PriorControlFactor=1
//         Observer: BandWidth=20
//   AXIS Axis102_54 P2M2_AndeviationY (id 102) // 2号叠片正极纠偏平台Y
//     Dynamic: Acceleration=11520, Deceleration=11520, Jerk=377018
//     Velo: Maximum=800
//     OtherSettings: AllowMotionCmdToSlave=true
//     encoder EncType=19
//       EncPara: ScaleFactorNumerator=5.96046e-07, MaxCount=#xffffffff
//     drive DrvType=16
//       DrvPara: MaxCount=#xffffffff, DriveControlDWord=#x00020100
//         Analog: VeloReferenz=800, TorqueSetpointScale=10, ScaleFactorActTorque=0.1
//         TimeComp: TaskDelayCycles=1
//     controller CtrType=1
//       CtrPara: PriorControlFactor=1
//         Observer: BandWidth=20
//   AXIS Axis103_55 P2M2_CaCarryingLine1 (id 103) // 2号叠片负极送片搬运1平移
//     Dynamic: Acceleration=47100, Deceleration=47100, Jerk=1297320
//     Velo: Maximum=3000
//     OtherSettings: AllowMotionCmdToSlave=true
//     encoder EncType=19
//       EncPara: MaxCount=#xffffffff
//     drive DrvType=16
//       DrvPara: MaxCount=#xffffffff, DriveControlDWord=#x00020100
//         Analog: VeloReferenz=3000, TorqueSetpointScale=10, ScaleFactorActTorque=0.1
//         TimeComp: TaskDelayCycles=1
//     controller CtrType=1
//       CtrPara: PriorControlFactor=1
//         Observer: BandWidth=20
//   AXIS Axis104_56 P2M2_CaCarryingUpDown1 (id 104) // 2号叠片负极送片搬运1升降
//     Dynamic: Acceleration=33500, Deceleration=33500, Jerk=3300740
//     Velo: Maximum=1000
//     OtherSettings: AllowMotionCmdToSlave=true
//     encoder EncType=19
//       EncPara: ScaleFactorNumerator=2.38419e-06, MaxCount=#xffffffff
//     drive DrvType=16
//       DrvPara: MaxCount=#xffffffff, DriveControlDWord=#x00020100
//         Analog: VeloReferenz=1000, TorqueSetpointScale=10, ScaleFactorActTorque=0.1
//         TimeComp: TaskDelayCycles=1
//     controller CtrType=1
//       CtrPara: PriorControlFactor=1
//         PosDiffControl: Enable=false
//         Observer: BandWidth=20
//   AXIS Axis105_57 P2M2_CaCarryingWhirling1 (id 105) // 2号叠片负极送片搬运1旋转
//     General: UnitName=°
//     Dynamic: Acceleration=189600, Deceleration=189600, Jerk=5164970
//     Velo: Maximum=12000
//     OtherSettings: AllowMotionCmdToSlave=true
//     encoder EncType=19
//       EncPara: ScaleFactorNumerator=2.86102e-05, MaxCount=#xffffffff
//     drive DrvType=16
//       DrvPara: MaxCount=#xffffffff, DriveControlDWord=#x00020100
//         Analog: VeloReferenz=12000, TorqueSetpointScale=10, ScaleFactorActTorque=0.1
//         TimeComp: TaskDelayCycles=1
//     controller CtrType=1
//       CtrPara: PriorControlFactor=1
//         PosDiffControl: Enable=false
//         Observer: BandWidth=20
//   AXIS Axis106_58 P2M2_CaCarryingLine2 (id 106) // 2号叠片负极送片搬运2平移
//     Dynamic: Acceleration=47100, Deceleration=47100, Jerk=1297320
//     Velo: Maximum=3000
//     OtherSettings: AllowMotionCmdToSlave=true
//     encoder EncType=19
//       EncPara: MaxCount=#xffffffff
//     drive DrvType=16
//       DrvPara: MaxCount=#xffffffff, DriveControlDWord=#x00020100
//         Analog: VeloReferenz=3000, TorqueSetpointScale=10, ScaleFactorActTorque=0.1
//         TimeComp: TaskDelayCycles=1
//     controller CtrType=1
//       CtrPara: PriorControlFactor=1
//         Observer: BandWidth=20
//   AXIS Axis107_59 P2M2_CaCarryingUpDown2 (id 107) // 2号叠片负极送片搬运2升降
//     Dynamic: Acceleration=15800, Deceleration=15800, Jerk=430414
//     Velo: Maximum=1000
//     OtherSettings: AllowMotionCmdToSlave=true
//     encoder EncType=19
//       EncPara: ScaleFactorNumerator=2.38419e-06, MaxCount=#xffffffff
//     drive DrvType=16
//       DrvPara: MaxCount=#xffffffff, DriveControlDWord=#x00020100
//         Analog: VeloReferenz=1000, TorqueSetpointScale=10, ScaleFactorActTorque=0.1
//         TimeComp: TaskDelayCycles=1
//     controller CtrType=1
//       CtrPara: PriorControlFactor=1
//         PosDiffControl: Enable=false
//         Observer: BandWidth=20
//   AXIS Axis108_60 P2M2_CaBelt (id 108) // 2号叠片负极送片皮带
//     Dynamic: Acceleration=41385, Deceleration=41385, Jerk=1166300
//     Velo: Maximum=2670
//     OtherSettings: AllowMotionCmdToSlave=true
//     encoder EncType=19
//       EncPara: ScaleFactorNumerator=6.36662e-06, MaxCount=#xffffffff
//     drive DrvType=16
//       DrvPara: MaxCount=#xffffffff, DriveControlDWord=#x00020100
//         Analog: VeloReferenz=2670, TorqueSetpointScale=10, ScaleFactorActTorque=0.1
//         TimeComp: TaskDelayCycles=1
//     controller CtrType=1
//       CtrPara: PriorControlFactor=1
//         PosDiffControl: Enable=false
//         Observer: BandWidth=20
//   AXIS Axis109_61 P2M2_CaDTCarryingLine (id 109) // 2号叠片负极叠台搬运平移
//     Dynamic: Acceleration=46500, Deceleration=46500, Jerk=1310450
//     Velo: Maximum=3000
//     OtherSettings: AllowMotionCmdToSlave=true
//     encoder EncType=19
//       EncPara: MaxCount=#xffffffff
//     drive DrvType=16
//       DrvPara: MaxCount=#xffffffff, DriveControlDWord=#x00020100
//         Analog: VeloReferenz=3000, TorqueSetpointScale=10, ScaleFactorActTorque=0.1
//         TimeComp: TaskDelayCycles=1
//     controller CtrType=1
//       CtrPara: PriorControlFactor=1
//         Observer: BandWidth=20
//   AXIS Axis110_62 P2M2_CaDTCarryingUpDown (id 110) // 2号叠片负极叠台搬运升降
//     Dynamic: Acceleration=15600, Deceleration=15600, Jerk=434571
//     Velo: Maximum=1000
//     OtherSettings: AllowMotionCmdToSlave=true
//     encoder EncType=19
//       EncPara: ScaleFactorNumerator=2.38419e-06, MaxCount=#xffffffff
//     drive DrvType=16
//       DrvPara: MaxCount=#xffffffff, DriveControlDWord=#x00020100
//         Analog: VeloReferenz=1000, TorqueSetpointScale=10, ScaleFactorActTorque=0.1
//         TimeComp: TaskDelayCycles=1
//     controller CtrType=1
//       CtrPara: PriorControlFactor=1
//         PosDiffControl: Enable=false
//         Observer: BandWidth=20
//   AXIS Axis111_63 P2M2_CadeviationX1 (id 111) // 2号叠片负极纠偏平台X1
//     Dynamic: Acceleration=11280, Deceleration=11280, Jerk=387922
//     Velo: Maximum=800
//     OtherSettings: AllowMotionCmdToSlave=true
//     encoder EncType=19
//       EncPara: ScaleFactorNumerator=5.96046e-07, MaxCount=#xffffffff
//     drive DrvType=16
//       DrvPara: MaxCount=#xffffffff, DriveControlDWord=#x00020100
//         Analog: VeloReferenz=800, TorqueSetpointScale=10, ScaleFactorActTorque=0.1
//         TimeComp: TaskDelayCycles=1
//     controller CtrType=1
//       CtrPara: PriorControlFactor=1
//         Observer: BandWidth=20
//   AXIS Axis112_64 P2M2_CadeviationX2 (id 112) // 2号叠片负极纠偏平台X2
//     Dynamic: Acceleration=11280, Deceleration=11280, Jerk=387922
//     Velo: Maximum=800
//     OtherSettings: AllowMotionCmdToSlave=true
//     encoder EncType=19
//       EncPara: ScaleFactorNumerator=5.96046e-07, MaxCount=#xffffffff
//     drive DrvType=16
//       DrvPara: MaxCount=#xffffffff, DriveControlDWord=#x00020100
//         Analog: VeloReferenz=800, TorqueSetpointScale=10, ScaleFactorActTorque=0.1
//         TimeComp: TaskDelayCycles=1
//     controller CtrType=1
//       CtrPara: PriorControlFactor=1
//         Observer: BandWidth=20
//   AXIS Axis113_65 P2M2_CadeviationY (id 113) // 2号叠片负极纠偏平台Y
//     Dynamic: Acceleration=11360, Deceleration=11360, Jerk=384076
//     Velo: Maximum=800
//     OtherSettings: AllowMotionCmdToSlave=true
//     encoder EncType=19
//       EncPara: ScaleFactorNumerator=5.96046e-07, MaxCount=#xffffffff
//     drive DrvType=16
//       DrvPara: MaxCount=#xffffffff, DriveControlDWord=#x00020100
//         Analog: VeloReferenz=800, TorqueSetpointScale=10, ScaleFactorActTorque=0.1
//         TimeComp: TaskDelayCycles=1
//     controller CtrType=1
//       CtrPara: PriorControlFactor=1
//         Observer: BandWidth=20
//   AXIS Axis114_66 P2M2_SEPTAunwinding (id 114) // 2号叠片隔膜放卷
//     General: UnitName=°
//     Dynamic: Acceleration=55440, Deceleration=55440, Jerk=1581070
//     Velo: Maximum=3600
//     OtherSettings: AllowMotionCmdToSlave=true
//     encoder EncType=19
//       EncPara: ScaleFactorNumerator=8.58307e-06, MaxCount=#xffffffff
//     drive DrvType=16
//       DrvPara: MaxCount=#xffffffff, DriveControlDWord=#x00020100
//         Analog: VeloReferenz=3600, TorqueSetpointScale=10, ScaleFactorActTorque=0.1
//         TimeComp: TaskDelayCycles=1
//     controller CtrType=1
//       CtrPara: PriorControlFactor=1
//         PosDiffControl: Enable=false
//         Observer: BandWidth=20
//   AXIS Axis115_67 P2M2_SEPTAdeviation1 (id 115) // 2号叠片隔膜放卷纠偏
//     Dynamic: Acceleration=3060, Deceleration=3060, Jerk=88335.8
//     Velo: Maximum=200
//     OtherSettings: AllowMotionCmdToSlave=true
//     encoder EncType=19
//       EncPara: ScaleFactorNumerator=4.76837e-07, MaxCount=#xffffffff
//     drive DrvType=16
//       DrvPara: MaxCount=#xffffffff, DriveControlDWord=#x00020100
//         Analog: VeloReferenz=200, TorqueSetpointScale=10, ScaleFactorActTorque=0.1
//         TimeComp: TaskDelayCycles=1
//     controller CtrType=1
//       CtrPara: PriorControlFactor=1
//         Observer: BandWidth=20
//   AXIS Axis116_68 P2M2_SEPTAdeviation2 (id 116) // 2号叠片隔膜尾部纠偏
//     Dynamic: Acceleration=3925, Deceleration=3925, Jerk=108110
//     Velo: Maximum=250
//     OtherSettings: AllowMotionCmdToSlave=true
//     encoder EncType=19
//       EncPara: ScaleFactorNumerator=5.96046e-07, MaxCount=#xffffffff
//     drive DrvType=16
//       DrvPara: MaxCount=#xffffffff, DriveControlDWord=#x00020100
//         Analog: VeloReferenz=250, TorqueSetpointScale=10, ScaleFactorActTorque=0.1
//         TimeComp: TaskDelayCycles=1
//     controller CtrType=1
//       CtrPara: PriorControlFactor=1
//         Observer: BandWidth=20
//   AXIS Axis117_69 P2M2_SEPTATension (id 117) // 2号叠片隔膜摆杆张力
//     General: UnitName=°
//     Velo: Maximum=18000
//     OtherSettings: AllowMotionCmdToSlave=true
//     encoder EncType=19
//       EncPara: ScaleFactorNumerator=4.29153e-05, MaxCount=#xffffffff
//     drive DrvType=16
//       DrvPara: MaxCount=#xffffffff, DriveControlDWord=#x00020000
//         Analog: VeloReferenz=18000, TorqueSetpointScale=10, ScaleFactorActTorque=0.1
//         TimeComp: TaskDelayCycles=1
//     controller CtrType=1
//       CtrPara: PriorControlFactor=1
//         PosDiffControl: Enable=false
//         Observer: BandWidth=20
//   AXIS Axis118_70 P2M2_SEPTATCache (id 118) // 2号叠片隔膜缓存
//     Dynamic: Acceleration=45600, Deceleration=45600, Jerk=1332920
//     Velo: Maximum=3000
//     OtherSettings: AllowMotionCmdToSlave=true
//     encoder EncType=19
//       EncPara: MaxCount=#xffffffff
//     drive DrvType=16
//       DrvPara: MaxCount=#xffffffff, DriveControlDWord=#x00020100
//         Analog: VeloReferenz=3000, TorqueSetpointScale=10, ScaleFactorActTorque=0.1
//         TimeComp: TaskDelayCycles=1
//     controller CtrType=1
//       CtrPara: PriorControlFactor=1
//         Observer: BandWidth=20
//   AXIS Axis119_71 P2M2_SEPTATLine (id 119) // 2号叠片隔膜平移
//     Dynamic: Acceleration=45300, Deceleration=45300, Jerk=1341240
//     Velo: Maximum=3000
//     OtherSettings: AllowMotionCmdToSlave=true
//     encoder EncType=19
//       EncPara: MaxCount=#xffffffff
//     drive DrvType=16
//       DrvPara: MaxCount=#xffffffff, DriveControlDWord=#x00020100
//         Analog: VeloReferenz=3000, TorqueSetpointScale=10, ScaleFactorActTorque=0.1
//         TimeComp: TaskDelayCycles=1
//     controller CtrType=1
//       CtrPara: PriorControlFactor=1
//         Observer: BandWidth=20
//   AXIS Axis120_72 P2M2_DTUpDownt (id 120) // 2号叠片叠台升降
//     Dynamic: Acceleration=3875, Deceleration=3875, Jerk=109205
//     Velo: Maximum=250
//     OtherSettings: AllowMotionCmdToSlave=true
//     encoder EncType=19
//       EncPara: ScaleFactorNumerator=5.96046e-07, MaxCount=#xffffffff
//     drive DrvType=16
//       DrvPara: MaxCount=#xffffffff, DriveControlDWord=#x00020100
//         Analog: VeloReferenz=250, TorqueSetpointScale=10, ScaleFactorActTorque=0.1
//         TimeComp: TaskDelayCycles=1
//     controller CtrType=1
//       CtrPara: PriorControlFactor=1
//         PosDiffControl: Enable=false
//         Observer: BandWidth=20
//   AXIS Axis121_73 P2M2_LeftYDLine (id 121) // 2号叠片左压刀开合
//     Dynamic: Acceleration=31600, Deceleration=31600, Jerk=860830
//     OtherSettings: AllowMotionCmdToSlave=true
//     encoder EncType=19
//       EncPara: ScaleFactorNumerator=1.3113e-05, MaxCount=#xffffffff
//     drive DrvType=16
//       DrvPara: MaxCount=#xffffffff, DriveControlDWord=#x00020100
//         Analog: VeloReferenz=5500, TorqueSetpointScale=10, ScaleFactorActTorque=0.1
//         TimeComp: TaskDelayCycles=1
//     controller CtrType=1
//       CtrPara: PriorControlFactor=1
//         PosDiffControl: Enable=false
//         Observer: BandWidth=20
//   AXIS Axis122_74 P2M2_LeftYDUpDown (id 122) // 2号叠片左压刀升降
//     Dynamic: Acceleration=3975, Deceleration=3975, Jerk=107123
//     Velo: Maximum=250
//     OtherSettings: AllowMotionCmdToSlave=true
//     encoder EncType=19
//       EncPara: ScaleFactorNumerator=5.96046e-07, MaxCount=#xffffffff
//     drive DrvType=16
//       DrvPara: MaxCount=#xffffffff, DriveControlDWord=#x00020100
//         Analog: VeloReferenz=250, TorqueSetpointScale=10, ScaleFactorActTorque=0.1
//         TimeComp: TaskDelayCycles=1
//     controller CtrType=1
//       CtrPara: PriorControlFactor=1
//         PosDiffControl: Enable=false
//         Observer: BandWidth=20
//   AXIS Axis123_75 P2M2_RightYDLine (id 123) // 2号叠片右压刀开合
//     Dynamic: Acceleration=31200, Deceleration=31200, Jerk=869143
//     OtherSettings: AllowMotionCmdToSlave=true
//     encoder EncType=19
//       EncPara: ScaleFactorNumerator=1.3113e-05, MaxCount=#xffffffff
//     drive DrvType=16
//       DrvPara: MaxCount=#xffffffff, DriveControlDWord=#x00020100
//         Analog: VeloReferenz=5500, TorqueSetpointScale=10, ScaleFactorActTorque=0.1
//         TimeComp: TaskDelayCycles=1
//     controller CtrType=1
//       CtrPara: PriorControlFactor=1
//         PosDiffControl: Enable=false
//         Observer: BandWidth=20
//   AXIS Axis124_76 P2M2_RightYDUpDown (id 124) // 2号叠片右压刀升降
//     Dynamic: Acceleration=3900, Deceleration=3900, Jerk=108643
//     Velo: Maximum=250
//     OtherSettings: AllowMotionCmdToSlave=true
//     encoder EncType=19
//       EncPara: ScaleFactorNumerator=5.96046e-07, MaxCount=#xffffffff
//     drive DrvType=16
//       DrvPara: MaxCount=#xffffffff, DriveControlDWord=#x00020100
//         Analog: VeloReferenz=250, TorqueSetpointScale=10, ScaleFactorActTorque=0.1
//         TimeComp: TaskDelayCycles=1
//     controller CtrType=1
//       CtrPara: PriorControlFactor=1
//         PosDiffControl: Enable=false
//         Observer: BandWidth=20
//   AXIS Axis125_77 P2M2_TailCurlLine (id 125) // 2号叠片尾卷夹电芯平移
//     Dynamic: Acceleration=2232, Deceleration=2232, Jerk=12580.4
//     Velo: Maximum=720
//     OtherSettings: AllowMotionCmdToSlave=true
//     encoder EncType=19
//       EncPara: ScaleFactorNumerator=1.72191e-06, MaxCount=#xffffffff
//     drive DrvType=16
//       DrvPara: MaxCount=#xffffffff, DriveControlDWord=#x00020100
//         Analog: VeloReferenz=720, TorqueSetpointScale=10, ScaleFactorActTorque=0.1
//         TimeComp: TaskDelayCycles=1
//     controller CtrType=1
//       CtrPara: PriorControlFactor=1
//         PosDiffControl: Enable=false
//         Observer: BandWidth=20
//   AXIS Axis126_78 P2M2_TailCurlUpDown (id 126) // 2号叠片尾卷夹电芯升降
//     Dynamic: Acceleration=3900, Deceleration=3900, Jerk=108643
//     Velo: Maximum=250
//     OtherSettings: AllowMotionCmdToSlave=true
//     encoder EncType=19
//       EncPara: ScaleFactorNumerator=5.96046e-07, MaxCount=#xffffffff
//     drive DrvType=16
//       DrvPara: MaxCount=#xffffffff, DriveControlDWord=#x00020100
//         Analog: VeloReferenz=250, TorqueSetpointScale=10, ScaleFactorActTorque=0.1
//         TimeComp: TaskDelayCycles=1
//     controller CtrType=1
//       CtrPara: PriorControlFactor=1
//         PosDiffControl: Enable=false
//         Observer: BandWidth=20
//   AXIS Axis127_79 P2M2_TailCurlRetracting (id 127) // 2号叠片尾卷夹电芯伸缩
//     Dynamic: Acceleration=70200, Deceleration=70200, Jerk=1955570
//     Velo: Maximum=4500
//     OtherSettings: AllowMotionCmdToSlave=true
//     encoder EncType=19
//       EncPara: ScaleFactorNumerator=1.07288e-05, MaxCount=#xffffffff
//     drive DrvType=16
//       DrvPara: MaxCount=#xffffffff, DriveControlDWord=#x00020100
//         Analog: VeloReferenz=4500, TorqueSetpointScale=10, ScaleFactorActTorque=0.1
//         TimeComp: TaskDelayCycles=1
//     controller CtrType=1
//       CtrPara: PriorControlFactor=1
//         PosDiffControl: Enable=false
//         Observer: BandWidth=20
//   AXIS Axis128_80 P2M2_TailCurlWhirling (id 128) // 2号叠片尾卷夹电芯旋转
//     General: UnitName=°
//     Dynamic: Acceleration=13590, Deceleration=13590, Jerk=402371
//     Velo: Maximum=900
//     OtherSettings: AllowMotionCmdToSlave=true
//     encoder EncType=19
//       EncPara: ScaleFactorNumerator=2.14577e-06, Offset=-3.433232e-05, MaxCount=#xffffffff, ReferenceSystem=1
//     drive DrvType=16
//       DrvPara: MaxCount=#xffffffff, DriveControlDWord=#x00020100
//         Analog: VeloReferenz=900, TorqueSetpointScale=10, ScaleFactorActTorque=0.1
//         TimeComp: TaskDelayCycles=1
//     controller CtrType=1
//       CtrPara: PriorControlFactor=1
//         PosDiffControl: Enable=false
//         Observer: BandWidth=20
//   AXIS Axis129_81 P2M2_TailCurlSEPTALine (id 129) // 2号叠片夹膜平移
//     Dynamic: Acceleration=11304, Deceleration=11304, Jerk=311356
//     Velo: Maximum=720
//     OtherSettings: AllowMotionCmdToSlave=true
//     encoder EncType=19
//       EncPara: ScaleFactorNumerator=1.72191e-06, Offset=-0.0002066292, MaxCount=#xffffffff, ReferenceSystem=1
//     drive DrvType=16
//       DrvPara: MaxCount=#xffffffff, DriveControlDWord=#x00020100
//         Analog: VeloReferenz=720, TorqueSetpointScale=10, ScaleFactorActTorque=0.1
//         TimeComp: TaskDelayCycles=1
//     controller CtrType=1
//       CtrPara: PriorControlFactor=1
//         PosDiffControl: Enable=false
//         Observer: BandWidth=20
//   AXIS Axis130_82 P2M2_TailCurlSEPTAUpDown (id 130) // 2号叠片夹膜升降
//     Dynamic: Acceleration=3900, Deceleration=3900, Jerk=108643
//     Velo: Maximum=250
//     OtherSettings: AllowMotionCmdToSlave=true
//     encoder EncType=19
//       EncPara: ScaleFactorNumerator=5.96046e-07, MaxCount=#xffffffff
//     drive DrvType=16
//       DrvPara: MaxCount=#xffffffff, DriveControlDWord=#x00020100
//         Analog: VeloReferenz=250, TorqueSetpointScale=10, ScaleFactorActTorque=0.1
//         TimeComp: TaskDelayCycles=1
//     controller CtrType=1
//       CtrPara: PriorControlFactor=1
//         PosDiffControl: Enable=false
//         Observer: BandWidth=20
//   AXIS Axis131_83 P2M2_LCurlingneedleLine (id 131) // 2号叠片长卷针平移
//     Dynamic: Acceleration=20280, Deceleration=20280, Jerk=564943
//     Velo: Maximum=1300
//     OtherSettings: AllowMotionCmdToSlave=true
//     encoder EncType=19
//       EncPara: ScaleFactorNumerator=0.01, MaxCount=#xffffffff
//     drive DrvType=16
//       DrvPara: MaxCount=#xffffffff, DriveControlDWord=#x00020000
//         Analog: VeloReferenz=1300, TorqueSetpointScale=10, ScaleFactorActTorque=0.1
//         TimeComp: TaskDelayCycles=1
//     controller CtrType=1
//       CtrPara: PriorControlFactor=1
//         PosDiffControl: Enable=false
//         Observer: BandWidth=20
//   AXIS Axis132_84 P2M2_SCurlingneedleLine (id 132) // 2号叠片短卷针平移
//     Dynamic: Acceleration=20280, Deceleration=20280, Jerk=564943
//     Velo: Maximum=1300
//     OtherSettings: AllowMotionCmdToSlave=true
//     encoder EncType=19
//       EncPara: ScaleFactorNumerator=0.01, MaxCount=#xffffffff
//     drive DrvType=16
//       DrvPara: MaxCount=#xffffffff, DriveControlDWord=#x00020000
//         Analog: VeloReferenz=1300, TorqueSetpointScale=10, ScaleFactorActTorque=0.1
//         TimeComp: TaskDelayCycles=1
//     controller CtrType=1
//       CtrPara: PriorControlFactor=1
//         PosDiffControl: Enable=false
//         Observer: BandWidth=20
//   AXIS Axis133_85 P2M2_LCurlingneedleWhirling (id 133) // 2号叠片长卷针旋转
//     General: UnitName=°, UnitFlags=#x00000004
//     Dynamic: Acceleration=36960, Deceleration=36960, Jerk=1054040
//     Velo: Maximum=2400
//     OtherSettings: AllowMotionCmdToSlave=true
//     encoder EncType=19
//       EncPara: ScaleFactorNumerator=0.018, MaxCount=#xffffffff
//     drive DrvType=16
//       DrvPara: MaxCount=#xffffffff, DriveControlDWord=#x00020000
//         Analog: VeloReferenz=2400, TorqueSetpointScale=10, ScaleFactorActTorque=0.1
//         TimeComp: TaskDelayCycles=1
//     controller CtrType=1
//       CtrPara: PriorControlFactor=1
//         PosDiffControl: Enable=false
//         Observer: BandWidth=20
//   AXIS Axis134_86 P2M2_SCurlingneedleWhirling (id 134) // 2号叠片短卷针旋转
//     General: UnitName=°, UnitFlags=#x00000004
//     Dynamic: Acceleration=37200, Deceleration=37200, Jerk=1048360
//     Velo: Maximum=2400
//     OtherSettings: AllowMotionCmdToSlave=true
//     encoder EncType=19
